LIN {X 0,Y 306.218,Z 83.638,A -85,B 0,C 180,E1 15314.136,E2 15314.136} C_VEL
LIN {X 0,Y 306.221,Z 83.636,A -85,B 0,C 180,E1 15309.585,E2 15309.585} C_VEL
LIN {X 0,Y 306.232,Z 83.637,A -85,B 0,C 180,E1 15305.245,E2 15305.245} C_VEL
LIN {X 0,Y 306.224,Z 83.64,A -85,B 0,C 180,E1 15300.748,E2 15300.748} C_VEL
LIN {X 0,Y 306.21,Z 83.649,A -85,B 0,C 180,E1 15296.255,E2 15296.255} C_VEL
LIN {X 0,Y 306.226,Z 83.648,A -85,B 0,C 180,E1 15291.74,E2 15291.74} C_VEL
LIN {X 0,Y 306.224,Z 83.645,A -85,B 0,C 180,E1 15287.171,E2 15287.171} C_VEL
LIN {X 0,Y 306.206,Z 83.645,A -85,B 0,C 180,E1 15282.713,E2 15282.713} C_VEL
LIN {X 0,Y 306.211,Z 83.626,A -85,B 0,C 180,E1 15278.146,E2 15278.146} C_VEL
LIN {X 0,Y 306.227,Z 83.646,A -85,B 0,C 180,E1 15273.637,E2 15273.637} C_VEL
LIN {X 0,Y 306.201,Z 83.621,A -85,B 0,C 180,E1 15269.158,E2 15269.158} C_VEL
LIN {X 0,Y 306.198,Z 83.63,A -85,B 0,C 180,E1 15264.691,E2 15264.691} C_VEL
LIN {X 0,Y 306.254,Z 83.929,A -85,B 0,C 180,E1 15261.619,E2 15261.619} C_VEL
LIN {X 0,Y 307.429,Z 87.023,A -85,B 0,C 180,E1 15260.879,E2 15260.879} C_VEL
LIN {X 0,Y 312.046,Z 96.934,A -85,B 0,C 180,E1 15258.694,E2 15258.694} C_VEL
LIN {X 0,Y 317.804,Z 111.108,A -85,B 0,C 180,E1 15255.831,E2 15255.831} C_VEL
LIN {X 0,Y 322.826,Z 126.337,A -85,B 0,C 180,E1 15253.034,E2 15253.034} C_VEL
LIN {X 0,Y 325.376,Z 136.231,A -85,B 0,C 180,E1 15251.349,E2 15251.349} C_VEL
LIN {X 0,Y 323.736,Z 169.935,A -85,B 0,C 180,E1 15247.17,E2 15247.17} C_VEL
LIN {X 0,Y 322.19,Z 205.367,A -85,B 0,C 180,E1 15242.891,E2 15242.891} C_VEL
LIN {X 0,Y 322.186,Z 209.699,A -85,B 0,C 180,E1 15242.451,E2 15242.451} C_VEL
LIN {X 0,Y 322.798,Z 215.074,A -85,B 0,C 180,E1 15242.253,E2 15242.253} C_VEL
LIN {X 0,Y 320.257,Z 311.161,A -85,B 0,C 180,E1 15240.104,E2 15240.104} C_VEL
LIN {X 0,Y 320.153,Z 327.939,A -85,B 0,C 180,E1 15239.578,E2 15239.578} C_VEL
LIN {X 0,Y 319.58,Z 341.902,A -85,B 0,C 180,E1 15238.832,E2 15238.832} C_VEL
LIN {X 0,Y 318.545,Z 355.587,A -85,B 0,C 180,E1 15237.78,E2 15237.78} C_VEL
LIN {X 0,Y 317.068,Z 368.764,A -85,B 0,C 180,E1 15236.398,E2 15236.398} C_VEL
LIN {X 0,Y 315.473,Z 380.218,A -85,B 0,C 180,E1 15234.829,E2 15234.829} C_VEL
LIN {X 0,Y 313.629,Z 391.275,A -85,B 0,C 180,E1 15232.887,E2 15232.887} C_VEL
LIN {X 0,Y 311.744,Z 401.04,A -85,B 0,C 180,E1 15230.657,E2 15230.657} C_VEL
LIN {X 0,Y 310.021,Z 409.095,A -85,B 0,C 180,E1 15228.229,E2 15228.229} C_VEL
LIN {X 0,Y 308.649,Z 415.111,A -85,B 0,C 180,E1 15225.788,E2 15225.788} C_VEL
LIN {X 0,Y 307.543,Z 419.693,A -85,B 0,C 180,E1 15223.153,E2 15223.153} C_VEL
LIN {X 0,Y 306.711,Z 422.772,A -85,B 0,C 180,E1 15220.137,E2 15220.137} C_VEL
LIN {X 0,Y 306.28,Z 423.761,A -85,B 0,C 180,E1 15217.124,E2 15217.124} C_VEL
LIN {X 0,Y 306.204,Z 422.716,A -85,B 0,C 180,E1 15214.118,E2 15214.118} C_VEL
LIN {X 0,Y 306.447,Z 419.874,A -85,B 0,C 180,E1 15211.307,E2 15211.307} C_VEL
LIN {X 0,Y 306.968,Z 415.503,A -85,B 0,C 180,E1 15208.692,E2 15208.692} C_VEL
LIN {X 0,Y 307.795,Z 409.247,A -85,B 0,C 180,E1 15206.087,E2 15206.087} C_VEL
LIN {X 0,Y 308.953,Z 400.726,A -85,B 0,C 180,E1 15203.495,E2 15203.495} C_VEL
LIN {X 0,Y 310.21,Z 391.122,A -85,B 0,C 180,E1 15201.286,E2 15201.286} C_VEL
LIN {X 0,Y 311.494,Z 380.394,A -85,B 0,C 180,E1 15199.363,E2 15199.363} C_VEL
LIN {X 0,Y 312.685,Z 368.716,A -85,B 0,C 180,E1 15197.721,E2 15197.721} C_VEL
LIN {X 0,Y 313.807,Z 355.087,A -85,B 0,C 180,E1 15196.267,E2 15196.267} C_VEL
LIN {X 0,Y 314.647,Z 340.308,A -85,B 0,C 180,E1 15195.13,E2 15195.13} C_VEL
LIN {X 0,Y 315.034,Z 325.009,A -85,B 0,C 180,E1 15194.342,E2 15194.342} C_VEL
LIN {X 0,Y 315.24,Z 322.674,A -85,B 0,C 180,E1 15194.17,E2 15194.17} C_VEL
LIN {X 0,Y 316.013,Z 321.401,A -85,B 0,C 180,E1 15193.879,E2 15193.879} C_VEL
LIN {X 0,Y 316.94,Z 321.781,A -85,B 0,C 180,E1 15193.693,E2 15193.693} C_VEL
LIN {X 0,Y 319.234,Z 322.708,A -85,B 0,C 180,E1 15193.439,E2 15193.439} C_VEL
LIN {X 0,Y 317.966,Z 338.659,A -85,B 0,C 180,E1 15192.327,E2 15192.327} C_VEL
LIN {X 0,Y 316.409,Z 352.982,A -85,B 0,C 180,E1 15191.004,E2 15191.004} C_VEL
LIN {X 0,Y 314.606,Z 366.938,A -85,B 0,C 180,E1 15189.342,E2 15189.342} C_VEL
LIN {X 0,Y 312.817,Z 379.43,A -85,B 0,C 180,E1 15187.445,E2 15187.445} C_VEL
LIN {X 0,Y 311.381,Z 388.653,A -85,B 0,C 180,E1 15185.723,E2 15185.723} C_VEL
LIN {X 0,Y 309.626,Z 393.761,A -85,B 0,C 180,E1 15184.686,E2 15184.686} C_VEL
LIN {X 0,Y 303.524,Z 403.055,A -85,B 0,C 180,E1 15182.617,E2 15182.617} C_VEL
LIN {X 0,Y 300.836,Z 407.741,A -85,B 0,C 180,E1 15181.279,E2 15181.279} C_VEL
LIN {X 0,Y 300.384,Z 409.36,A -85,B 0,C 180,E1 15180.736,E2 15180.736} C_VEL
LIN {X 0,Y 299.326,Z 416.103,A -85,B 0,C 180,E1 15177.918,E2 15177.918} C_VEL
LIN {X 0,Y 298.675,Z 420.99,A -85,B 0,C 180,E1 15175.078,E2 15175.078} C_VEL
LIN {X 0,Y 298.375,Z 424.115,A -85,B 0,C 180,E1 15172.175,E2 15172.175} C_VEL
LIN {X 0,Y 298.432,Z 425.598,A -85,B 0,C 180,E1 15169.206,E2 15169.206} C_VEL
LIN {X 0,Y 298.87,Z 425.294,A -85,B 0,C 180,E1 15166.17,E2 15166.17} C_VEL
LIN {X 0,Y 299.771,Z 423.124,A -85,B 0,C 180,E1 15163.074,E2 15163.074} C_VEL
LIN {X 0,Y 301.067,Z 419.248,A -85,B 0,C 180,E1 15160.195,E2 15160.195} C_VEL
LIN {X 0,Y 302.907,Z 413.394,A -85,B 0,C 180,E1 15157.295,E2 15157.295} C_VEL
LIN {X 0,Y 305.079,Z 405.985,A -85,B 0,C 180,E1 15154.651,E2 15154.651} C_VEL
LIN {X 0,Y 307.546,Z 397.131,A -85,B 0,C 180,E1 15152.221,E2 15152.221} C_VEL
LIN {X 0,Y 310.231,Z 386.618,A -85,B 0,C 180,E1 15149.971,E2 15149.971} C_VEL
LIN {X 0,Y 313.092,Z 374.223,A -85,B 0,C 180,E1 15147.885,E2 15147.885} C_VEL
LIN {X 0,Y 315.783,Z 360.648,A -85,B 0,C 180,E1 15146.112,E2 15146.112} C_VEL
LIN {X 0,Y 318.084,Z 346.959,A -85,B 0,C 180,E1 15144.709,E2 15144.709} C_VEL
LIN {X 0,Y 320.126,Z 331.5,A -85,B 0,C 180,E1 15143.512,E2 15143.512} C_VEL
LIN {X 0,Y 321.698,Z 315.374,A -85,B 0,C 180,E1 15142.606,E2 15142.606} C_VEL
LIN {X 0,Y 322.948,Z 294.587,A -85,B 0,C 180,E1 15141.877,E2 15141.877} C_VEL
LIN {X 0,Y 327.686,Z 217.917,A -85,B 0,C 180,E1 15139.693,E2 15139.693} C_VEL
LIN {X 0,Y 323.711,Z 190.896,A -85,B 0,C 180,E1 15138.038,E2 15138.038} C_VEL
LIN {X 0,Y 320.283,Z 171.007,A -85,B 0,C 180,E1 15136.585,E2 15136.585} C_VEL
LIN {X 0,Y 323.837,Z 155.783,A -85,B 0,C 180,E1 15133.663,E2 15133.663} C_VEL
LIN {X 0,Y 321.635,Z 144.592,A -85,B 0,C 180,E1 15130.388,E2 15130.388} C_VEL
LIN {X 0,Y 319.074,Z 134.629,A -85,B 0,C 180,E1 15127.02,E2 15127.02} C_VEL
LIN {X 0,Y 316.628,Z 126.45,A -85,B 0,C 180,E1 15123.803,E2 15123.803} C_VEL
LIN {X 0,Y 314.2,Z 119.063,A -85,B 0,C 180,E1 15120.365,E2 15120.365} C_VEL
LIN {X 0,Y 312.239,Z 114.196,A -85,B 0,C 180,E1 15117.567,E2 15117.567} C_VEL
LIN {X 0,Y 311.17,Z 111.425,A -85,B 0,C 180,E1 15115.762,E2 15115.762} C_VEL
LIN {X 0,Y 309.858,Z 108.044,A -85,B 0,C 180,E1 15113.143,E2 15113.143} C_VEL
LIN {X 0,Y 308.302,Z 104.197,A -85,B 0,C 180,E1 15108.969,E2 15108.969} C_VEL
LIN {X 0,Y 307.15,Z 102.355,A -85,B 0,C 180,E1 15103.937,E2 15103.937} C_VEL
LIN {X 0,Y 307.285,Z 102.523,A -85,B 0,C 180,E1 15100.023,E2 15100.023} C_VEL
LIN {X 0,Y 308.962,Z 104.848,A -85,B 0,C 180,E1 15094.917,E2 15094.917} C_VEL
LIN {X 0,Y 311.201,Z 109.842,A -85,B 0,C 180,E1 15090.345,E2 15090.345} C_VEL
LIN {X 0,Y 313.233,Z 114.532,A -85,B 0,C 180,E1 15087.354,E2 15087.354} C_VEL
LIN {X 0,Y 315.016,Z 118.627,A -85,B 0,C 180,E1 15085.158,E2 15085.158} C_VEL
LIN {X 0,Y 317.64,Z 124.79,A -85,B 0,C 180,E1 15082.362,E2 15082.362} C_VEL
LIN {X 0,Y 321.226,Z 134.301,A -85,B 0,C 180,E1 15078.874,E2 15078.874} C_VEL
LIN {X 0,Y 324.75,Z 144.909,A -85,B 0,C 180,E1 15075.662,E2 15075.662} C_VEL
LIN {X 0,Y 328.156,Z 157.046,A -85,B 0,C 180,E1 15072.565,E2 15072.565} C_VEL
LIN {X 0,Y 328.381,Z 158.338,A -85,B 0,C 180,E1 15072.278,E2 15072.278} C_VEL
LIN {X 0,Y 326.983,Z 164.325,A -85,B 0,C 180,E1 15071.492,E2 15071.492} C_VEL
LIN {X 0,Y 329.661,Z 192.112,A -85,B 0,C 180,E1 15070.189,E2 15070.189} C_VEL
LIN {X 0,Y 329.69,Z 198.596,A -85,B 0,C 180,E1 15069.987,E2 15069.987} C_VEL
LIN {X 0,Y 324.108,Z 330.652,A -85,B 0,C 180,E1 15067,E2 15067} C_VEL
LIN {X 0,Y 322.996,Z 351.571,A -85,B 0,C 180,E1 15066.447,E2 15066.447} C_VEL
LIN {X 0,Y 321.026,Z 369.794,A -85,B 0,C 180,E1 15065.677,E2 15065.677} C_VEL
LIN {X 0,Y 318.428,Z 386.883,A -85,B 0,C 180,E1 15064.635,E2 15064.635} C_VEL
LIN {X 0,Y 315.355,Z 403.595,A -85,B 0,C 180,E1 15063.266,E2 15063.266} C_VEL
LIN {X 0,Y 311.891,Z 420.167,A -85,B 0,C 180,E1 15061.504,E2 15061.504} C_VEL
LIN {X 0,Y 308.53,Z 435.036,A -85,B 0,C 180,E1 15059.512,E2 15059.512} C_VEL
LIN {X 0,Y 305.249,Z 448.999,A -85,B 0,C 180,E1 15057.191,E2 15057.191} C_VEL
LIN {X 0,Y 302.216,Z 462.009,A -85,B 0,C 180,E1 15054.521,E2 15054.521} C_VEL
LIN {X 0,Y 299.688,Z 473.731,A -85,B 0,C 180,E1 15051.532,E2 15051.532} C_VEL
LIN {X 0,Y 297.903,Z 483.696,A -85,B 0,C 180,E1 15048.392,E2 15048.392} C_VEL
LIN {X 0,Y 296.829,Z 492.632,A -85,B 0,C 180,E1 15044.834,E2 15044.834} C_VEL
LIN {X 0,Y 296.583,Z 499.123,A -85,B 0,C 180,E1 15041.474,E2 15041.474} C_VEL
LIN {X 0,Y 296.941,Z 504.12,A -85,B 0,C 180,E1 15037.937,E2 15037.937} C_VEL
LIN {X 0,Y 297.552,Z 507.104,A -85,B 0,C 180,E1 15034.627,E2 15034.627} C_VEL
LIN {X 0,Y 298.008,Z 508.377,A -85,B 0,C 180,E1 15031.539,E2 15031.539} C_VEL
LIN {X 0,Y 298.055,Z 508.203,A -85,B 0,C 180,E1 15028.656,E2 15028.656} C_VEL
LIN {X 0,Y 297.673,Z 506.535,A -85,B 0,C 180,E1 15025.571,E2 15025.571} C_VEL
LIN {X 0,Y 297.132,Z 503.314,A -85,B 0,C 180,E1 15022.461,E2 15022.461} C_VEL
LIN {X 0,Y 296.743,Z 498.122,A -85,B 0,C 180,E1 15019.125,E2 15019.125} C_VEL
LIN {X 0,Y 296.849,Z 491.021,A -85,B 0,C 180,E1 15015.768,E2 15015.768} C_VEL
LIN {X 0,Y 297.621,Z 481.81,A -85,B 0,C 180,E1 15012.403,E2 15012.403} C_VEL
LIN {X 0,Y 298.972,Z 471.647,A -85,B 0,C 180,E1 15009.444,E2 15009.444} C_VEL
LIN {X 0,Y 300.853,Z 460.093,A -85,B 0,C 180,E1 15006.706,E2 15006.706} C_VEL
LIN {X 0,Y 303.17,Z 447.087,A -85,B 0,C 180,E1 15004.195,E2 15004.195} C_VEL
LIN {X 0,Y 305.808,Z 432.438,A -85,B 0,C 180,E1 15001.915,E2 15001.915} C_VEL
LIN {X 0,Y 308.392,Z 417.575,A -85,B 0,C 180,E1 15000.049,E2 15000.049} C_VEL
LIN {X 0,Y 311.025,Z 401.011,A -85,B 0,C 180,E1 14998.401,E2 14998.401} C_VEL
LIN {X 0,Y 313.395,Z 383.904,A -85,B 0,C 180,E1 14997.097,E2 14997.097} C_VEL
LIN {X 0,Y 315.377,Z 366.084,A -85,B 0,C 180,E1 14996.106,E2 14996.106} C_VEL
LIN {X 0,Y 316.7,Z 347.608,A -85,B 0,C 180,E1 14995.417,E2 14995.417} C_VEL
LIN {X 0,Y 322.005,Z 178.475,A -85,B 0,C 180,E1 14991.663,E2 14991.663} C_VEL
LIN {X 0,Y 321.492,Z 158.885,A -85,B 0,C 180,E1 14991.083,E2 14991.083} C_VEL
LIN {X 0,Y 323.297,Z 143.638,A -85,B 0,C 180,E1 14989.9,E2 14989.9} C_VEL
LIN {X 0,Y 314.968,Z 122.157,A -85,B 0,C 180,E1 14986.897,E2 14986.897} C_VEL
LIN {X 0,Y 306.931,Z 103.52,A -85,B 0,C 180,E1 14983.937,E2 14983.937} C_VEL
LIN {X 0,Y 299.48,Z 87.935,A -85,B 0,C 180,E1 14981.125,E2 14981.125} C_VEL
LIN {X 0,Y 298.366,Z 85.034,A -85,B 0,C 180,E1 14980.55,E2 14980.55} C_VEL
LIN {X 0,Y 298.295,Z 84.644,A -85,B 0,C 180,E1 14979.808,E2 14979.808} C_VEL
LIN {X 0,Y 298.29,Z 84.632,A -85,B 0,C 180,E1 14975.131,E2 14975.131} C_VEL
LIN {X 0,Y 298.304,Z 84.636,A -85,B 0,C 180,E1 14970.529,E2 14970.529} C_VEL
LIN {X 0,Y 298.288,Z 84.642,A -85,B 0,C 180,E1 14966.047,E2 14966.047} C_VEL
LIN {X 0,Y 298.289,Z 84.641,A -85,B 0,C 180,E1 14961.43,E2 14961.43} C_VEL
LIN {X 0,Y 298.297,Z 84.64,A -85,B 0,C 180,E1 14956.954,E2 14956.954} C_VEL
LIN {X 0,Y 298.29,Z 84.638,A -85,B 0,C 180,E1 14952.584,E2 14952.584} C_VEL
LIN {X 0,Y 298.279,Z 84.638,A -85,B 0,C 180,E1 14947.899,E2 14947.899} C_VEL
LIN {X 0,Y 298.29,Z 84.633,A -85,B 0,C 180,E1 14943.266,E2 14943.266} C_VEL
LIN {X 0,Y 298.286,Z 84.628,A -85,B 0,C 180,E1 14938.847,E2 14938.847} C_VEL
LIN {X 0,Y 298.27,Z 84.632,A -85,B 0,C 180,E1 14934.228,E2 14934.228} C_VEL
LIN {X 0,Y 298.282,Z 84.628,A -85,B 0,C 180,E1 14929.766,E2 14929.766} C_VEL
LIN {X 0,Y 298.29,Z 84.629,A -85,B 0,C 180,E1 14925.241,E2 14925.241} C_VEL
LIN {X 0,Y 298.267,Z 84.64,A -85,B 0,C 180,E1 14920.617,E2 14920.617} C_VEL
LIN {X 0,Y 298.275,Z 84.594,A -85,B 0,C 180,E1 14916.07,E2 14916.07} C_VEL
LIN {X 0,Y 298.285,Z 84.622,A -85,B 0,C 180,E1 14911.576,E2 14911.576} C_VEL
LIN {X 0,Y 298.263,Z 84.646,A -85,B 0,C 180,E1 14907.107,E2 14907.107} C_VEL
LIN {X 0,Y 298.285,Z 84.823,A -85,B 0,C 180,E1 14903.05,E2 14903.05} C_VEL
LIN {X 0,Y 299.159,Z 87.431,A -85,B 0,C 180,E1 14902.379,E2 14902.379} C_VEL
LIN {X 0,Y 300.565,Z 90.006,A -85,B 0,C 180,E1 14901.724,E2 14901.724} C_VEL
LIN {X 0,Y 306.143,Z 102.165,A -85,B 0,C 180,E1 14898.969,E2 14898.969} C_VEL
LIN {X 0,Y 311.601,Z 115.952,A -85,B 0,C 180,E1 14896.124,E2 14896.124} C_VEL
LIN {X 0,Y 316.602,Z 131.405,A -85,B 0,C 180,E1 14893.257,E2 14893.257} C_VEL
LIN {X 0,Y 318.588,Z 138.968,A -85,B 0,C 180,E1 14891.943,E2 14891.943} C_VEL
LIN {X 0,Y 316.728,Z 174.086,A -85,B 0,C 180,E1 14887.534,E2 14887.534} C_VEL
LIN {X 0,Y 315.112,Z 210.08,A -85,B 0,C 180,E1 14883.186,E2 14883.186} C_VEL
LIN {X 0,Y 315.824,Z 216.202,A -85,B 0,C 180,E1 14882.945,E2 14882.945} C_VEL
LIN {X 0,Y 313.162,Z 311.56,A -85,B 0,C 180,E1 14880.769,E2 14880.769} C_VEL
LIN {X 0,Y 313.042,Z 328.708,A -85,B 0,C 180,E1 14880.227,E2 14880.227} C_VEL
LIN {X 0,Y 312.47,Z 342.308,A -85,B 0,C 180,E1 14879.498,E2 14879.498} C_VEL
LIN {X 0,Y 311.3,Z 356.975,A -85,B 0,C 180,E1 14878.35,E2 14878.35} C_VEL
LIN {X 0,Y 309.679,Z 370.641,A -85,B 0,C 180,E1 14876.871,E2 14876.871} C_VEL
LIN {X 0,Y 307.907,Z 382.491,A -85,B 0,C 180,E1 14875.174,E2 14875.174} C_VEL
LIN {X 0,Y 306.065,Z 392.819,A -85,B 0,C 180,E1 14873.282,E2 14873.282} C_VEL
LIN {X 0,Y 304.091,Z 402.488,A -85,B 0,C 180,E1 14871,E2 14871} C_VEL
LIN {X 0,Y 302.286,Z 410.469,A -85,B 0,C 180,E1 14868.512,E2 14868.512} C_VEL
LIN {X 0,Y 300.748,Z 416.791,A -85,B 0,C 180,E1 14865.818,E2 14865.818} C_VEL
LIN {X 0,Y 299.61,Z 421.153,A -85,B 0,C 180,E1 14863.115,E2 14863.115} C_VEL
LIN {X 0,Y 298.805,Z 423.925,A -85,B 0,C 180,E1 14860.214,E2 14860.214} C_VEL
LIN {X 0,Y 298.354,Z 424.856,A -85,B 0,C 180,E1 14857.121,E2 14857.121} C_VEL
LIN {X 0,Y 298.28,Z 423.753,A -85,B 0,C 180,E1 14854.035,E2 14854.035} C_VEL
LIN {X 0,Y 298.542,Z 420.842,A -85,B 0,C 180,E1 14851.15,E2 14851.15} C_VEL
LIN {X 0,Y 299.097,Z 416.397,A -85,B 0,C 180,E1 14848.466,E2 14848.466} C_VEL
LIN {X 0,Y 299.977,Z 410.066,A -85,B 0,C 180,E1 14845.793,E2 14845.793} C_VEL
LIN {X 0,Y 301.102,Z 402.148,A -85,B 0,C 180,E1 14843.324,E2 14843.324} C_VEL
LIN {X 0,Y 302.41,Z 392.647,A -85,B 0,C 180,E1 14841.059,E2 14841.059} C_VEL
LIN {X 0,Y 303.748,Z 382.05,A -85,B 0,C 180,E1 14839.088,E2 14839.088} C_VEL
LIN {X 0,Y 305.064,Z 369.787,A -85,B 0,C 180,E1 14837.314,E2 14837.314} C_VEL
LIN {X 0,Y 306.24,Z 356.15,A -85,B 0,C 180,E1 14835.825,E2 14835.825} C_VEL
LIN {X 0,Y 307.124,Z 341.358,A -85,B 0,C 180,E1 14834.661,E2 14834.661} C_VEL
LIN {X 0,Y 307.553,Z 332.982,A -85,B 0,C 180,E1 14834.107,E2 14834.107} C_VEL
LIN {X 0,Y 308.443,Z 331.887,A -85,B 0,C 180,E1 14833.763,E2 14833.763} C_VEL
LIN {X 0,Y 311.174,Z 333.159,A -85,B 0,C 180,E1 14833.355,E2 14833.355} C_VEL
LIN {X 0,Y 309.531,Z 348.896,A -85,B 0,C 180,E1 14832.009,E2 14832.009} C_VEL
LIN {X 0,Y 307.639,Z 363.677,A -85,B 0,C 180,E1 14830.352,E2 14830.352} C_VEL
LIN {X 0,Y 305.596,Z 377.731,A -85,B 0,C 180,E1 14828.301,E2 14828.301} C_VEL
LIN {X 0,Y 303.681,Z 389.594,A -85,B 0,C 180,E1 14826.088,E2 14826.088} C_VEL
LIN {X 0,Y 301.964,Z 399.884,A -85,B 0,C 180,E1 14823.659,E2 14823.659} C_VEL
LIN {X 0,Y 300.472,Z 408.792,A -85,B 0,C 180,E1 14820.932,E2 14820.932} C_VEL
LIN {X 0,Y 300.384,Z 409.36,A -85,B 0,C 180,E1 14820.736,E2 14820.736} C_VEL
LIN {X 0,Y 298.873,Z 412.989,A -85,B 0,C 180,E1 14819.453,E2 14819.453} C_VEL
LIN {X 0,Y 294.088,Z 418.356,A -85,B 0,C 180,E1 14817.258,E2 14817.258} C_VEL
LIN {X 0,Y 291.155,Z 421.554,A -85,B 0,C 180,E1 14815.481,E2 14815.481} C_VEL
LIN {X 0,Y 290.67,Z 422.702,A -85,B 0,C 180,E1 14814.639,E2 14814.639} C_VEL
LIN {X 0,Y 290.43,Z 425.743,A -85,B 0,C 180,E1 14811.454,E2 14811.454} C_VEL
LIN {X 0,Y 290.597,Z 426.821,A -85,B 0,C 180,E1 14808.3,E2 14808.3} C_VEL
LIN {X 0,Y 291.176,Z 426.156,A -85,B 0,C 180,E1 14805.255,E2 14805.255} C_VEL
LIN {X 0,Y 292.151,Z 423.829,A -85,B 0,C 180,E1 14802.332,E2 14802.332} C_VEL
LIN {X 0,Y 293.674,Z 419.566,A -85,B 0,C 180,E1 14799.292,E2 14799.292} C_VEL
LIN {X 0,Y 295.672,Z 413.576,A -85,B 0,C 180,E1 14796.405,E2 14796.405} C_VEL
LIN {X 0,Y 298.186,Z 405.572,A -85,B 0,C 180,E1 14793.592,E2 14793.592} C_VEL
LIN {X 0,Y 300.902,Z 396.224,A -85,B 0,C 180,E1 14791.101,E2 14791.101} C_VEL
LIN {X 0,Y 303.732,Z 385.585,A -85,B 0,C 180,E1 14788.877,E2 14788.877} C_VEL
LIN {X 0,Y 306.49,Z 374.05,A -85,B 0,C 180,E1 14786.966,E2 14786.966} C_VEL
LIN {X 0,Y 309.467,Z 359.746,A -85,B 0,C 180,E1 14785.102,E2 14785.102} C_VEL
LIN {X 0,Y 311.913,Z 345.474,A -85,B 0,C 180,E1 14783.672,E2 14783.672} C_VEL
LIN {X 0,Y 314.095,Z 329.395,A -85,B 0,C 180,E1 14782.458,E2 14782.458} C_VEL
LIN {X 0,Y 315.67,Z 312.422,A -85,B 0,C 180,E1 14781.569,E2 14781.569} C_VEL
LIN {X 0,Y 317.627,Z 281.324,A -85,B 0,C 180,E1 14780.578,E2 14780.578} C_VEL
LIN {X 0,Y 321.613,Z 219.163,A -85,B 0,C 180,E1 14778.782,E2 14778.782} C_VEL
LIN {X 0,Y 317.859,Z 192.52,A -85,B 0,C 180,E1 14777.081,E2 14777.081} C_VEL
LIN {X 0,Y 314.18,Z 170.966,A -85,B 0,C 180,E1 14775.455,E2 14775.455} C_VEL
LIN {X 0,Y 317.08,Z 159.096,A -85,B 0,C 180,E1 14773.123,E2 14773.123} C_VEL
LIN {X 0,Y 315.055,Z 148.38,A -85,B 0,C 180,E1 14769.868,E2 14769.868} C_VEL
LIN {X 0,Y 312.512,Z 138.076,A -85,B 0,C 180,E1 14766.245,E2 14766.245} C_VEL
LIN {X 0,Y 309.93,Z 129.366,A -85,B 0,C 180,E1 14762.589,E2 14762.589} C_VEL
LIN {X 0,Y 307.785,Z 123.166,A -85,B 0,C 180,E1 14759.442,E2 14759.442} C_VEL
LIN {X 0,Y 306.027,Z 117.882,A -85,B 0,C 180,E1 14756.254,E2 14756.254} C_VEL
LIN {X 0,Y 304.313,Z 113.734,A -85,B 0,C 180,E1 14752.87,E2 14752.87} C_VEL
LIN {X 0,Y 302.929,Z 110.091,A -85,B 0,C 180,E1 14748.771,E2 14748.771} C_VEL
LIN {X 0,Y 301.922,Z 108.386,A -85,B 0,C 180,E1 14743.651,E2 14743.651} C_VEL
LIN {X 0,Y 302.176,Z 108.736,A -85,B 0,C 180,E1 14739.67,E2 14739.67} C_VEL
LIN {X 0,Y 303.784,Z 111.056,A -85,B 0,C 180,E1 14734.841,E2 14734.841} C_VEL
LIN {X 0,Y 305.898,Z 115.909,A -85,B 0,C 180,E1 14730.396,E2 14730.396} C_VEL
LIN {X 0,Y 307.724,Z 120.203,A -85,B 0,C 180,E1 14727.58,E2 14727.58} C_VEL
LIN {X 0,Y 309.665,Z 124.824,A -85,B 0,C 180,E1 14725.098,E2 14725.098} C_VEL
LIN {X 0,Y 312.169,Z 131.034,A -85,B 0,C 180,E1 14722.283,E2 14722.283} C_VEL
LIN {X 0,Y 315.429,Z 139.952,A -85,B 0,C 180,E1 14718.976,E2 14718.976} C_VEL
LIN {X 0,Y 318.791,Z 150.454,A -85,B 0,C 180,E1 14715.746,E2 14715.746} C_VEL
LIN {X 0,Y 321.704,Z 161.505,A -85,B 0,C 180,E1 14712.896,E2 14712.896} C_VEL
LIN {X 0,Y 321.066,Z 164.544,A -85,B 0,C 180,E1 14712.516,E2 14712.516} C_VEL
LIN {X 0,Y 323.554,Z 191.512,A -85,B 0,C 180,E1 14711.182,E2 14711.182} C_VEL
LIN {X 0,Y 323.746,Z 198.251,A -85,B 0,C 180,E1 14710.934,E2 14710.934} C_VEL
LIN {X 0,Y 316.998,Z 346.321,A -85,B 0,C 180,E1 14707.479,E2 14707.479} C_VEL
LIN {X 0,Y 315.136,Z 364.811,A -85,B 0,C 180,E1 14706.754,E2 14706.754} C_VEL
LIN {X 0,Y 312.668,Z 381.422,A -85,B 0,C 180,E1 14705.818,E2 14705.818} C_VEL
LIN {X 0,Y 309.617,Z 398.158,A -85,B 0,C 180,E1 14704.536,E2 14704.536} C_VEL
LIN {X 0,Y 306.226,Z 414.206,A -85,B 0,C 180,E1 14702.933,E2 14702.933} C_VEL
LIN {X 0,Y 302.687,Z 429.303,A -85,B 0,C 180,E1 14701.019,E2 14701.019} C_VEL
LIN {X 0,Y 299.026,Z 443.988,A -85,B 0,C 180,E1 14698.675,E2 14698.675} C_VEL
LIN {X 0,Y 295.724,Z 457.159,A -85,B 0,C 180,E1 14696.076,E2 14696.076} C_VEL
LIN {X 0,Y 292.831,Z 469.263,A -85,B 0,C 180,E1 14693.121,E2 14693.121} C_VEL
LIN {X 0,Y 290.623,Z 479.85,A -85,B 0,C 180,E1 14689.915,E2 14689.915} C_VEL
LIN {X 0,Y 289.191,Z 488.934,A -85,B 0,C 180,E1 14686.471,E2 14686.471} C_VEL
LIN {X 0,Y 288.614,Z 496.386,A -85,B 0,C 180,E1 14682.811,E2 14682.811} C_VEL
LIN {X 0,Y 288.785,Z 501.85,A -85,B 0,C 180,E1 14679.166,E2 14679.166} C_VEL
LIN {X 0,Y 289.391,Z 505.332,A -85,B 0,C 180,E1 14675.704,E2 14675.704} C_VEL
LIN {X 0,Y 289.953,Z 507.042,A -85,B 0,C 180,E1 14672.571,E2 14672.571} C_VEL
LIN {X 0,Y 290.173,Z 507.299,A -85,B 0,C 180,E1 14669.607,E2 14669.607} C_VEL
LIN {X 0,Y 289.911,Z 506.154,A -85,B 0,C 180,E1 14666.64,E2 14666.64} C_VEL
LIN {X 0,Y 289.357,Z 503.445,A -85,B 0,C 180,E1 14663.454,E2 14663.454} C_VEL
LIN {X 0,Y 288.847,Z 498.832,A -85,B 0,C 180,E1 14660.035,E2 14660.035} C_VEL
LIN {X 0,Y 288.794,Z 492.358,A -85,B 0,C 180,E1 14656.589,E2 14656.589} C_VEL
LIN {X 0,Y 289.371,Z 483.918,A -85,B 0,C 180,E1 14653.159,E2 14653.159} C_VEL
LIN {X 0,Y 290.585,Z 474.343,A -85,B 0,C 180,E1 14650.086,E2 14650.086} C_VEL
LIN {X 0,Y 292.48,Z 462.627,A -85,B 0,C 180,E1 14647.065,E2 14647.065} C_VEL
LIN {X 0,Y 294.735,Z 450.263,A -85,B 0,C 180,E1 14644.472,E2 14644.472} C_VEL
LIN {X 0,Y 297.436,Z 435.961,A -85,B 0,C 180,E1 14642.037,E2 14642.037} C_VEL
LIN {X 0,Y 300.257,Z 420.604,A -85,B 0,C 180,E1 14639.936,E2 14639.936} C_VEL
LIN {X 0,Y 302.929,Z 404.953,A -85,B 0,C 180,E1 14638.236,E2 14638.236} C_VEL
LIN {X 0,Y 305.378,Z 388.657,A -85,B 0,C 180,E1 14636.856,E2 14636.856} C_VEL
LIN {X 0,Y 307.602,Z 370.716,A -85,B 0,C 180,E1 14635.735,E2 14635.735} C_VEL
LIN {X 0,Y 309.172,Z 352.612,A -85,B 0,C 180,E1 14634.956,E2 14634.956} C_VEL
LIN {X 0,Y 310.134,Z 327.851,A -85,B 0,C 180,E1 14634.322,E2 14634.322} C_VEL
LIN {X 0,Y 315.038,Z 179.291,A -85,B 0,C 180,E1 14630.971,E2 14630.971} C_VEL
LIN {X 0,Y 314.622,Z 158.089,A -85,B 0,C 180,E1 14630.302,E2 14630.302} C_VEL
LIN {X 0,Y 316.097,Z 146.113,A -85,B 0,C 180,E1 14629.34,E2 14629.34} C_VEL
LIN {X 0,Y 307.764,Z 124.504,A -85,B 0,C 180,E1 14626.215,E2 14626.215} C_VEL
LIN {X 0,Y 299.01,Z 104.371,A -85,B 0,C 180,E1 14622.881,E2 14622.881} C_VEL
LIN {X 0,Y 291.934,Z 89.484,A -85,B 0,C 180,E1 14620.082,E2 14620.082} C_VEL
LIN {X 0,Y 290.433,Z 86.152,A -85,B 0,C 180,E1 14619.388,E2 14619.388} C_VEL
LIN {X 0,Y 290.362,Z 85.623,A -85,B 0,C 180,E1 14618.905,E2 14618.905} C_VEL
LIN {X 0,Y 290.357,Z 85.625,A -85,B 0,C 180,E1 14614.145,E2 14614.145} C_VEL
LIN {X 0,Y 290.351,Z 85.63,A -85,B 0,C 180,E1 14609.402,E2 14609.402} C_VEL
LIN {X 0,Y 290.358,Z 85.623,A -85,B 0,C 180,E1 14604.841,E2 14604.841} C_VEL
LIN {X 0,Y 290.351,Z 85.624,A -85,B 0,C 180,E1 14600.353,E2 14600.353} C_VEL
LIN {X 0,Y 290.344,Z 85.624,A -85,B 0,C 180,E1 14595.581,E2 14595.581} C_VEL
LIN {X 0,Y 290.354,Z 85.623,A -85,B 0,C 180,E1 14590.917,E2 14590.917} C_VEL
LIN {X 0,Y 290.339,Z 85.627,A -85,B 0,C 180,E1 14586.326,E2 14586.326} C_VEL
LIN {X 0,Y 290.348,Z 85.628,A -85,B 0,C 180,E1 14581.578,E2 14581.578} C_VEL
LIN {X 0,Y 290.347,Z 85.63,A -85,B 0,C 180,E1 14576.989,E2 14576.989} C_VEL
LIN {X 0,Y 290.332,Z 85.632,A -85,B 0,C 180,E1 14572.281,E2 14572.281} C_VEL
LIN {X 0,Y 290.348,Z 85.628,A -85,B 0,C 180,E1 14567.672,E2 14567.672} C_VEL
LIN {X 0,Y 290.343,Z 85.625,A -85,B 0,C 180,E1 14563.185,E2 14563.185} C_VEL
LIN {X 0,Y 290.324,Z 85.611,A -85,B 0,C 180,E1 14558.588,E2 14558.588} C_VEL
LIN {X 0,Y 290.342,Z 85.611,A -85,B 0,C 180,E1 14553.997,E2 14553.997} C_VEL
LIN {X 0,Y 290.344,Z 85.592,A -85,B 0,C 180,E1 14549.587,E2 14549.587} C_VEL
LIN {X 0,Y 290.32,Z 85.62,A -85,B 0,C 180,E1 14544.89,E2 14544.89} C_VEL
LIN {X 0,Y 290.402,Z 86.088,A -85,B 0,C 180,E1 14544.417,E2 14544.417} C_VEL
LIN {X 0,Y 292.148,Z 89.784,A -85,B 0,C 180,E1 14543.451,E2 14543.451} C_VEL
LIN {X 0,Y 297.834,Z 101.678,A -85,B 0,C 180,E1 14540.542,E2 14540.542} C_VEL
LIN {X 0,Y 303.541,Z 115.56,A -85,B 0,C 180,E1 14537.525,E2 14537.525} C_VEL
LIN {X 0,Y 308.446,Z 129.845,A -85,B 0,C 180,E1 14534.7,E2 14534.7} C_VEL
LIN {X 0,Y 311.807,Z 142.278,A -85,B 0,C 180,E1 14532.478,E2 14532.478} C_VEL
LIN {X 0,Y 309.768,Z 178.097,A -85,B 0,C 180,E1 14527.941,E2 14527.941} C_VEL
LIN {X 0,Y 308.184,Z 211.152,A -85,B 0,C 180,E1 14523.917,E2 14523.917} C_VEL
LIN {X 0,Y 308.902,Z 217.32,A -85,B 0,C 180,E1 14523.669,E2 14523.669} C_VEL
LIN {X 0,Y 306.111,Z 311.998,A -85,B 0,C 180,E1 14521.464,E2 14521.464} C_VEL
LIN {X 0,Y 305.974,Z 329.487,A -85,B 0,C 180,E1 14520.905,E2 14520.905} C_VEL
LIN {X 0,Y 305.34,Z 343.61,A -85,B 0,C 180,E1 14520.133,E2 14520.133} C_VEL
LIN {X 0,Y 304.113,Z 358.137,A -85,B 0,C 180,E1 14518.969,E2 14518.969} C_VEL
LIN {X 0,Y 302.415,Z 371.743,A -85,B 0,C 180,E1 14517.464,E2 14517.464} C_VEL
LIN {X 0,Y 300.55,Z 383.594,A -85,B 0,C 180,E1 14515.729,E2 14515.729} C_VEL
LIN {X 0,Y 298.707,Z 393.474,A -85,B 0,C 180,E1 14513.89,E2 14513.89} C_VEL
LIN {X 0,Y 296.612,Z 403.239,A -85,B 0,C 180,E1 14511.555,E2 14511.555} C_VEL
LIN {X 0,Y 294.688,Z 411.294,A -85,B 0,C 180,E1 14509.007,E2 14509.007} C_VEL
LIN {X 0,Y 293.144,Z 417.31,A -85,B 0,C 180,E1 14506.443,E2 14506.443} C_VEL
LIN {X 0,Y 291.895,Z 421.89,A -85,B 0,C 180,E1 14503.67,E2 14503.67} C_VEL
LIN {X 0,Y 290.943,Z 424.967,A -85,B 0,C 180,E1 14500.493,E2 14500.493} C_VEL
LIN {X 0,Y 290.446,Z 425.952,A -85,B 0,C 180,E1 14497.316,E2 14497.316} C_VEL
LIN {X 0,Y 290.347,Z 424.903,A -85,B 0,C 180,E1 14494.146,E2 14494.146} C_VEL
LIN {X 0,Y 290.608,Z 422.057,A -85,B 0,C 180,E1 14491.181,E2 14491.181} C_VEL
LIN {X 0,Y 291.179,Z 417.682,A -85,B 0,C 180,E1 14488.424,E2 14488.424} C_VEL
LIN {X 0,Y 292.087,Z 411.421,A -85,B 0,C 180,E1 14485.68,E2 14485.68} C_VEL
LIN {X 0,Y 293.36,Z 402.892,A -85,B 0,C 180,E1 14482.951,E2 14482.951} C_VEL
LIN {X 0,Y 294.74,Z 393.281,A -85,B 0,C 180,E1 14480.627,E2 14480.627} C_VEL
LIN {X 0,Y 296.148,Z 382.542,A -85,B 0,C 180,E1 14478.607,E2 14478.607} C_VEL
LIN {X 0,Y 297.458,Z 370.85,A -85,B 0,C 180,E1 14476.885,E2 14476.885} C_VEL
LIN {X 0,Y 298.698,Z 357.104,A -85,B 0,C 180,E1 14475.35,E2 14475.35} C_VEL
LIN {X 0,Y 299.815,Z 341.36,A -85,B 0,C 180,E1 14474.029,E2 14474.029} C_VEL
LIN {X 0,Y 300.709,Z 340.513,A -85,B 0,C 180,E1 14473.681,E2 14473.681} C_VEL
LIN {X 0,Y 303.031,Z 341.513,A -85,B 0,C 180,E1 14473.317,E2 14473.317} C_VEL
LIN {X 0,Y 301.235,Z 356.539,A -85,B 0,C 180,E1 14471.819,E2 14471.819} C_VEL
LIN {X 0,Y 299.308,Z 370.123,A -85,B 0,C 180,E1 14470.077,E2 14470.077} C_VEL
LIN {X 0,Y 297.183,Z 383.607,A -85,B 0,C 180,E1 14467.862,E2 14467.862} C_VEL
LIN {X 0,Y 295.237,Z 394.889,A -85,B 0,C 180,E1 14465.488,E2 14465.488} C_VEL
LIN {X 0,Y 293.554,Z 404.522,A -85,B 0,C 180,E1 14462.919,E2 14462.919} C_VEL
LIN {X 0,Y 292.119,Z 412.888,A -85,B 0,C 180,E1 14459.994,E2 14459.994} C_VEL
LIN {X 0,Y 291.172,Z 418.909,A -85,B 0,C 180,E1 14457.141,E2 14457.141} C_VEL
LIN {X 0,Y 290.67,Z 422.702,A -85,B 0,C 180,E1 14454.639,E2 14454.639} C_VEL
LIN {X 0,Y 289.517,Z 424.489,A -85,B 0,C 180,E1 14453.163,E2 14453.163} C_VEL
LIN {X 0,Y 285.191,Z 426.956,A -85,B 0,C 180,E1 14450.553,E2 14450.553} C_VEL
LIN {X 0,Y 282.905,Z 427.906,A -85,B 0,C 180,E1 14448.586,E2 14448.586} C_VEL
LIN {X 0,Y 282.746,Z 427.98,A -85,B 0,C 180,E1 14447.797,E2 14447.797} C_VEL
LIN {X 0,Y 283.381,Z 427.233,A -85,B 0,C 180,E1 14444.83,E2 14444.83} C_VEL
LIN {X 0,Y 284.582,Z 424.517,A -85,B 0,C 180,E1 14441.55,E2 14441.55} C_VEL
LIN {X 0,Y 286.303,Z 420.057,A -85,B 0,C 180,E1 14438.436,E2 14438.436} C_VEL
LIN {X 0,Y 288.625,Z 413.456,A -85,B 0,C 180,E1 14435.347,E2 14435.347} C_VEL
LIN {X 0,Y 291.259,Z 405.517,A -85,B 0,C 180,E1 14432.614,E2 14432.614} C_VEL
LIN {X 0,Y 294.358,Z 395.383,A -85,B 0,C 180,E1 14429.956,E2 14429.956} C_VEL
LIN {X 0,Y 297.277,Z 384.891,A -85,B 0,C 180,E1 14427.8,E2 14427.8} C_VEL
LIN {X 0,Y 300.582,Z 371.532,A -85,B 0,C 180,E1 14425.649,E2 14425.649} C_VEL
LIN {X 0,Y 303.398,Z 358.143,A -85,B 0,C 180,E1 14423.974,E2 14423.974} C_VEL
LIN {X 0,Y 305.997,Z 343.234,A -85,B 0,C 180,E1 14422.528,E2 14422.528} C_VEL
LIN {X 0,Y 308.075,Z 327.652,A -85,B 0,C 180,E1 14421.405,E2 14421.405} C_VEL
LIN {X 0,Y 309.667,Z 310.782,A -85,B 0,C 180,E1 14420.55,E2 14420.55} C_VEL
LIN {X 0,Y 315.489,Z 226.103,A -85,B 0,C 180,E1 14418.016,E2 14418.016} C_VEL
LIN {X 0,Y 315.671,Z 220.222,A -85,B 0,C 180,E1 14417.81,E2 14417.81} C_VEL
LIN {X 0,Y 312.063,Z 193.866,A -85,B 0,C 180,E1 14416.067,E2 14416.067} C_VEL
LIN {X 0,Y 308.245,Z 171.07,A -85,B 0,C 180,E1 14414.272,E2 14414.272} C_VEL
LIN {X 0,Y 310.335,Z 162.307,A -85,B 0,C 180,E1 14412.517,E2 14412.517} C_VEL
LIN {X 0,Y 308.369,Z 151.627,A -85,B 0,C 180,E1 14409.142,E2 14409.142} C_VEL
LIN {X 0,Y 306.1,Z 142.067,A -85,B 0,C 180,E1 14405.624,E2 14405.624} C_VEL
LIN {X 0,Y 303.799,Z 133.982,A -85,B 0,C 180,E1 14402.075,E2 14402.075} C_VEL
LIN {X 0,Y 301.606,Z 126.917,A -85,B 0,C 180,E1 14398.291,E2 14398.291} C_VEL
LIN {X 0,Y 299.892,Z 122.526,A -85,B 0,C 180,E1 14395.219,E2 14395.219} C_VEL
LIN {X 0,Y 298.839,Z 119.519,A -85,B 0,C 180,E1 14392.696,E2 14392.696} C_VEL
LIN {X 0,Y 297.637,Z 116.092,A -85,B 0,C 180,E1 14388.765,E2 14388.765} C_VEL
LIN {X 0,Y 296.713,Z 114.449,A -85,B 0,C 180,E1 14383.557,E2 14383.557} C_VEL
LIN {X 0,Y 297.04,Z 114.893,A -85,B 0,C 180,E1 14379.509,E2 14379.509} C_VEL
LIN {X 0,Y 298.556,Z 117.206,A -85,B 0,C 180,E1 14374.829,E2 14374.829} C_VEL
LIN {X 0,Y 300.573,Z 121.89,A -85,B 0,C 180,E1 14370.507,E2 14370.507} C_VEL
LIN {X 0,Y 302.256,Z 125.902,A -85,B 0,C 180,E1 14367.82,E2 14367.82} C_VEL
LIN {X 0,Y 304.121,Z 130.517,A -85,B 0,C 180,E1 14365.279,E2 14365.279} C_VEL
LIN {X 0,Y 306.536,Z 136.74,A -85,B 0,C 180,E1 14362.414,E2 14362.414} C_VEL
LIN {X 0,Y 309.47,Z 145.063,A -85,B 0,C 180,E1 14359.26,E2 14359.26} C_VEL
LIN {X 0,Y 312.644,Z 155.366,A -85,B 0,C 180,E1 14356.02,E2 14356.02} C_VEL
LIN {X 0,Y 315.17,Z 164.648,A -85,B 0,C 180,E1 14353.605,E2 14353.605} C_VEL
LIN {X 0,Y 317.325,Z 186.796,A -85,B 0,C 180,E1 14352.421,E2 14352.421} C_VEL
LIN {X 0,Y 317.943,Z 198.597,A -85,B 0,C 180,E1 14351.915,E2 14351.915} C_VEL
LIN {X 0,Y 311.737,Z 327.59,A -85,B 0,C 180,E1 14348.877,E2 14348.877} C_VEL
LIN {X 0,Y 310.46,Z 349.753,A -85,B 0,C 180,E1 14348.278,E2 14348.278} C_VEL
LIN {X 0,Y 308.368,Z 367.786,A -85,B 0,C 180,E1 14347.501,E2 14347.501} C_VEL
LIN {X 0,Y 305.529,Z 384.908,A -85,B 0,C 180,E1 14346.44,E2 14346.44} C_VEL
LIN {X 0,Y 302.17,Z 401.596,A -85,B 0,C 180,E1 14345.038,E2 14345.038} C_VEL
LIN {X 0,Y 298.34,Z 418.16,A -85,B 0,C 180,E1 14343.228,E2 14343.228} C_VEL
LIN {X 0,Y 294.618,Z 432.925,A -85,B 0,C 180,E1 14341.18,E2 14341.18} C_VEL
LIN {X 0,Y 290.906,Z 446.909,A -85,B 0,C 180,E1 14338.764,E2 14338.764} C_VEL
LIN {X 0,Y 287.47,Z 459.824,A -85,B 0,C 180,E1 14335.993,E2 14335.993} C_VEL
LIN {X 0,Y 284.601,Z 471.235,A -85,B 0,C 180,E1 14332.954,E2 14332.954} C_VEL
LIN {X 0,Y 282.439,Z 481.226,A -85,B 0,C 180,E1 14329.653,E2 14329.653} C_VEL
LIN {X 0,Y 281.034,Z 490.186,A -85,B 0,C 180,E1 14325.901,E2 14325.901} C_VEL
LIN {X 0,Y 280.606,Z 497.062,A -85,B 0,C 180,E1 14322.137,E2 14322.137} C_VEL
LIN {X 0,Y 280.931,Z 502.059,A -85,B 0,C 180,E1 14318.34,E2 14318.34} C_VEL
LIN {X 0,Y 281.599,Z 504.933,A -85,B 0,C 180,E1 14314.89,E2 14314.89} C_VEL
LIN {X 0,Y 282.147,Z 506.148,A -85,B 0,C 180,E1 14311.626,E2 14311.626} C_VEL
LIN {X 0,Y 282.225,Z 505.95,A -85,B 0,C 180,E1 14308.784,E2 14308.784} C_VEL
LIN {X 0,Y 281.806,Z 504.295,A -85,B 0,C 180,E1 14305.558,E2 14305.558} C_VEL
LIN {X 0,Y 281.191,Z 501.007,A -85,B 0,C 180,E1 14302.236,E2 14302.236} C_VEL
LIN {X 0,Y 280.792,Z 495.754,A -85,B 0,C 180,E1 14298.708,E2 14298.708} C_VEL
LIN {X 0,Y 280.961,Z 488.57,A -85,B 0,C 180,E1 14295.156,E2 14295.156} C_VEL
LIN {X 0,Y 281.81,Z 479.852,A -85,B 0,C 180,E1 14291.809,E2 14291.809} C_VEL
LIN {X 0,Y 283.314,Z 469.684,A -85,B 0,C 180,E1 14288.687,E2 14288.687} C_VEL
LIN {X 0,Y 285.388,Z 458.106,A -85,B 0,C 180,E1 14285.803,E2 14285.803} C_VEL
LIN {X 0,Y 287.931,Z 445.066,A -85,B 0,C 180,E1 14283.167,E2 14283.167} C_VEL
LIN {X 0,Y 290.804,Z 430.366,A -85,B 0,C 180,E1 14280.778,E2 14280.778} C_VEL
LIN {X 0,Y 293.602,Z 415.426,A -85,B 0,C 180,E1 14278.829,E2 14278.829} C_VEL
LIN {X 0,Y 296.451,Z 398.731,A -85,B 0,C 180,E1 14277.113,E2 14277.113} C_VEL
LIN {X 0,Y 298.979,Z 381.447,A -85,B 0,C 180,E1 14275.762,E2 14275.762} C_VEL
LIN {X 0,Y 301.081,Z 363.467,A -85,B 0,C 180,E1 14274.747,E2 14274.747} C_VEL
LIN {X 0,Y 302.385,Z 345.057,A -85,B 0,C 180,E1 14274.064,E2 14274.064} C_VEL
LIN {X 0,Y 308.086,Z 179.572,A -85,B 0,C 180,E1 14270.237,E2 14270.237} C_VEL
LIN {X 0,Y 307.66,Z 158.712,A -85,B 0,C 180,E1 14269.585,E2 14269.585} C_VEL
LIN {X 0,Y 308.929,Z 148.576,A -85,B 0,C 180,E1 14268.753,E2 14268.753} C_VEL
LIN {X 0,Y 301.026,Z 128.064,A -85,B 0,C 180,E1 14265.707,E2 14265.707} C_VEL
LIN {X 0,Y 292.911,Z 109.158,A -85,B 0,C 180,E1 14262.5,E2 14262.5} C_VEL
LIN {X 0,Y 285.664,Z 94.019,A -85,B 0,C 180,E1 14259.57,E2 14259.57} C_VEL
LIN {X 0,Y 282.509,Z 87.177,A -85,B 0,C 180,E1 14258.14,E2 14258.14} C_VEL
LIN {X 0,Y 282.415,Z 86.632,A -85,B 0,C 180,E1 14257.769,E2 14257.769} C_VEL
LIN {X 0,Y 282.418,Z 86.614,A -85,B 0,C 180,E1 14252.963,E2 14252.963} C_VEL
LIN {X 0,Y 282.423,Z 86.605,A -85,B 0,C 180,E1 14248.32,E2 14248.32} C_VEL
LIN {X 0,Y 282.408,Z 86.603,A -85,B 0,C 180,E1 14243.517,E2 14243.517} C_VEL
LIN {X 0,Y 282.42,Z 86.602,A -85,B 0,C 180,E1 14238.794,E2 14238.794} C_VEL
LIN {X 0,Y 282.4,Z 86.604,A -85,B 0,C 180,E1 14234.053,E2 14234.053} C_VEL
LIN {X 0,Y 282.409,Z 86.601,A -85,B 0,C 180,E1 14229.373,E2 14229.373} C_VEL
LIN {X 0,Y 282.411,Z 86.601,A -85,B 0,C 180,E1 14224.874,E2 14224.874} C_VEL
LIN {X 0,Y 282.395,Z 86.603,A -85,B 0,C 180,E1 14220.202,E2 14220.202} C_VEL
LIN {X 0,Y 282.407,Z 86.605,A -85,B 0,C 180,E1 14215.532,E2 14215.532} C_VEL
LIN {X 0,Y 282.405,Z 86.605,A -85,B 0,C 180,E1 14211.026,E2 14211.026} C_VEL
LIN {X 0,Y 282.39,Z 86.606,A -85,B 0,C 180,E1 14206.277,E2 14206.277} C_VEL
LIN {X 0,Y 282.411,Z 86.605,A -85,B 0,C 180,E1 14201.585,E2 14201.585} C_VEL
LIN {X 0,Y 282.387,Z 86.573,A -85,B 0,C 180,E1 14197.007,E2 14197.007} C_VEL
LIN {X 0,Y 282.401,Z 86.61,A -85,B 0,C 180,E1 14192.137,E2 14192.137} C_VEL
LIN {X 0,Y 282.405,Z 86.604,A -85,B 0,C 180,E1 14187.681,E2 14187.681} C_VEL
LIN {X 0,Y 282.446,Z 86.923,A -85,B 0,C 180,E1 14186.113,E2 14186.113} C_VEL
LIN {X 0,Y 283.921,Z 90.408,A -85,B 0,C 180,E1 14185.134,E2 14185.134} C_VEL
LIN {X 0,Y 284.968,Z 92.193,A -85,B 0,C 180,E1 14184.624,E2 14184.624} C_VEL
LIN {X 0,Y 290.844,Z 104.306,A -85,B 0,C 180,E1 14181.519,E2 14181.519} C_VEL
LIN {X 0,Y 296.578,Z 118.062,A -85,B 0,C 180,E1 14178.382,E2 14178.382} C_VEL
LIN {X 0,Y 301.404,Z 131.861,A -85,B 0,C 180,E1 14175.576,E2 14175.576} C_VEL
LIN {X 0,Y 305.085,Z 145.167,A -85,B 0,C 180,E1 14173.111,E2 14173.111} C_VEL
LIN {X 0,Y 302.964,Z 180.535,A -85,B 0,C 180,E1 14168.588,E2 14168.588} C_VEL
LIN {X 0,Y 301.336,Z 212.369,A -85,B 0,C 180,E1 14164.677,E2 14164.677} C_VEL
LIN {X 0,Y 302.031,Z 218.497,A -85,B 0,C 180,E1 14164.425,E2 14164.425} C_VEL
LIN {X 0,Y 299.109,Z 312.396,A -85,B 0,C 180,E1 14162.193,E2 14162.193} C_VEL
LIN {X 0,Y 298.951,Z 330.267,A -85,B 0,C 180,E1 14161.616,E2 14161.616} C_VEL
LIN {X 0,Y 298.305,Z 344.186,A -85,B 0,C 180,E1 14160.85,E2 14160.85} C_VEL
LIN {X 0,Y 297.012,Z 358.875,A -85,B 0,C 180,E1 14159.658,E2 14159.658} C_VEL
LIN {X 0,Y 295.294,Z 372.061,A -85,B 0,C 180,E1 14158.184,E2 14158.184} C_VEL
LIN {X 0,Y 293.433,Z 383.519,A -85,B 0,C 180,E1 14156.509,E2 14156.509} C_VEL
LIN {X 0,Y 291.383,Z 394.124,A -85,B 0,C 180,E1 14154.53,E2 14154.53} C_VEL
LIN {X 0,Y 289.066,Z 404.387,A -85,B 0,C 180,E1 14152.027,E2 14152.027} C_VEL
LIN {X 0,Y 286.976,Z 412.673,A -85,B 0,C 180,E1 14149.327,E2 14149.327} C_VEL
LIN {X 0,Y 285.247,Z 418.993,A -85,B 0,C 180,E1 14146.493,E2 14146.493} C_VEL
LIN {X 0,Y 283.951,Z 423.379,A -85,B 0,C 180,E1 14143.621,E2 14143.621} C_VEL
LIN {X 0,Y 283.039,Z 426.121,A -85,B 0,C 180,E1 14140.583,E2 14140.583} C_VEL
LIN {X 0,Y 282.52,Z 427.048,A -85,B 0,C 180,E1 14137.318,E2 14137.318} C_VEL
LIN {X 0,Y 282.422,Z 425.939,A -85,B 0,C 180,E1 14134.059,E2 14134.059} C_VEL
LIN {X 0,Y 282.704,Z 423.023,A -85,B 0,C 180,E1 14131.012,E2 14131.012} C_VEL
LIN {X 0,Y 283.312,Z 418.573,A -85,B 0,C 180,E1 14128.178,E2 14128.178} C_VEL
LIN {X 0,Y 284.279,Z 412.235,A -85,B 0,C 180,E1 14125.359,E2 14125.359} C_VEL
LIN {X 0,Y 285.517,Z 404.31,A -85,B 0,C 180,E1 14122.756,E2 14122.756} C_VEL
LIN {X 0,Y 286.953,Z 394.798,A -85,B 0,C 180,E1 14120.371,E2 14120.371} C_VEL
LIN {X 0,Y 288.422,Z 384.189,A -85,B 0,C 180,E1 14118.298,E2 14118.298} C_VEL
LIN {X 0,Y 289.87,Z 371.907,A -85,B 0,C 180,E1 14116.433,E2 14116.433} C_VEL
LIN {X 0,Y 291.161,Z 358.249,A -85,B 0,C 180,E1 14114.87,E2 14114.87} C_VEL
LIN {X 0,Y 291.941,Z 348.837,A -85,B 0,C 180,E1 14113.995,E2 14113.995} C_VEL
LIN {X 0,Y 292.797,Z 348.019,A -85,B 0,C 180,E1 14113.635,E2 14113.635} C_VEL
LIN {X 0,Y 294.882,Z 349.213,A -85,B 0,C 180,E1 14113.248,E2 14113.248} C_VEL
LIN {X 0,Y 292.767,Z 364.501,A -85,B 0,C 180,E1 14111.48,E2 14111.48} C_VEL
LIN {X 0,Y 290.645,Z 378.006,A -85,B 0,C 180,E1 14109.457,E2 14109.457} C_VEL
LIN {X 0,Y 288.694,Z 389.376,A -85,B 0,C 180,E1 14107.322,E2 14107.322} C_VEL
LIN {X 0,Y 286.772,Z 399.884,A -85,B 0,C 180,E1 14104.825,E2 14104.825} C_VEL
LIN {X 0,Y 285.195,Z 408.598,A -85,B 0,C 180,E1 14102.206,E2 14102.206} C_VEL
LIN {X 0,Y 283.88,Z 416.071,A -85,B 0,C 180,E1 14099.25,E2 14099.25} C_VEL
LIN {X 0,Y 283.042,Z 421.543,A -85,B 0,C 180,E1 14096.315,E2 14096.315} C_VEL
LIN {X 0,Y 282.564,Z 425.582,A -85,B 0,C 180,E1 14093.018,E2 14093.018} C_VEL
LIN {X 0,Y 282.541,Z 427.615,A -85,B 0,C 180,E1 14089.853,E2 14089.853} C_VEL
LIN {X 0,Y 282.746,Z 427.98,A -85,B 0,C 180,E1 14087.797,E2 14087.797} C_VEL
LIN {X 0,Y 282.062,Z 427.994,A -85,B 0,C 180,E1 14086.227,E2 14086.227} C_VEL
LIN {X 0,Y 278.608,Z 427.348,A -85,B 0,C 180,E1 14083.457,E2 14083.457} C_VEL
LIN {X 0,Y 276.998,Z 425.958,A -85,B 0,C 180,E1 14081.43,E2 14081.43} C_VEL
LIN {X 0,Y 277.111,Z 425.129,A -85,B 0,C 180,E1 14080.644,E2 14080.644} C_VEL
LIN {X 0,Y 278.99,Z 420.476,A -85,B 0,C 180,E1 14077.536,E2 14077.536} C_VEL
LIN {X 0,Y 281.456,Z 413.972,A -85,B 0,C 180,E1 14074.494,E2 14074.494} C_VEL
LIN {X 0,Y 284.33,Z 405.769,A -85,B 0,C 180,E1 14071.678,E2 14071.678} C_VEL
LIN {X 0,Y 287.442,Z 396.212,A -85,B 0,C 180,E1 14069.143,E2 14069.143} C_VEL
LIN {X 0,Y 290.524,Z 385.69,A -85,B 0,C 180,E1 14066.953,E2 14066.953} C_VEL
LIN {X 0,Y 294.01,Z 372.314,A -85,B 0,C 180,E1 14064.768,E2 14064.768} C_VEL
LIN {X 0,Y 297,Z 358.874,A -85,B 0,C 180,E1 14063.059,E2 14063.059} C_VEL
LIN {X 0,Y 299.792,Z 343.759,A -85,B 0,C 180,E1 14061.569,E2 14061.569} C_VEL
LIN {X 0,Y 301.971,Z 328.244,A -85,B 0,C 180,E1 14060.438,E2 14060.438} C_VEL
LIN {X 0,Y 303.636,Z 311.412,A -85,B 0,C 180,E1 14059.575,E2 14059.575} C_VEL
LIN {X 0,Y 309.814,Z 225.321,A -85,B 0,C 180,E1 14056.967,E2 14056.967} C_VEL
LIN {X 0,Y 309.818,Z 221.344,A -85,B 0,C 180,E1 14056.801,E2 14056.801} C_VEL
LIN {X 0,Y 306.503,Z 195.647,A -85,B 0,C 180,E1 14055.031,E2 14055.031} C_VEL
LIN {X 0,Y 302.455,Z 170.828,A -85,B 0,C 180,E1 14052.991,E2 14052.991} C_VEL
LIN {X 0,Y 303.702,Z 165.901,A -85,B 0,C 180,E1 14051.971,E2 14051.971} C_VEL
LIN {X 0,Y 301.899,Z 155.494,A -85,B 0,C 180,E1 14048.571,E2 14048.571} C_VEL
LIN {X 0,Y 299.789,Z 146.138,A -85,B 0,C 180,E1 14044.975,E2 14044.975} C_VEL
LIN {X 0,Y 297.521,Z 137.873,A -85,B 0,C 180,E1 14041.156,E2 14041.156} C_VEL
LIN {X 0,Y 295.617,Z 131.834,A -85,B 0,C 180,E1 14037.674,E2 14037.674} C_VEL
LIN {X 0,Y 294.263,Z 128.068,A -85,B 0,C 180,E1 14034.932,E2 14034.932} C_VEL
LIN {X 0,Y 293.39,Z 125.34,A -85,B 0,C 180,E1 14032.56,E2 14032.56} C_VEL
LIN {X 0,Y 292.293,Z 122.009,A -85,B 0,C 180,E1 14028.557,E2 14028.557} C_VEL
LIN {X 0,Y 291.504,Z 120.512,A -85,B 0,C 180,E1 14023.46,E2 14023.46} C_VEL
LIN {X 0,Y 291.851,Z 120.978,A -85,B 0,C 180,E1 14019.547,E2 14019.547} C_VEL
LIN {X 0,Y 293.289,Z 123.169,A -85,B 0,C 180,E1 14014.993,E2 14014.993} C_VEL
LIN {X 0,Y 295.167,Z 127.587,A -85,B 0,C 180,E1 14010.805,E2 14010.805} C_VEL
LIN {X 0,Y 296.87,Z 131.954,A -85,B 0,C 180,E1 14007.85,E2 14007.85} C_VEL
LIN {X 0,Y 298.695,Z 136.495,A -85,B 0,C 180,E1 14005.315,E2 14005.315} C_VEL
LIN {X 0,Y 301.474,Z 143.954,A -85,B 0,C 180,E1 14001.912,E2 14001.912} C_VEL
LIN {X 0,Y 304.533,Z 153.405,A -85,B 0,C 180,E1 13998.455,E2 13998.455} C_VEL
LIN {X 0,Y 307.485,Z 164.025,A -85,B 0,C 180,E1 13995.251,E2 13995.251} C_VEL
LIN {X 0,Y 310.053,Z 169.496,A -85,B 0,C 180,E1 13994.425,E2 13994.425} C_VEL
LIN {X 0,Y 312.176,Z 196.196,A -85,B 0,C 180,E1 13993.04,E2 13993.04} C_VEL
LIN {X 0,Y 311.797,Z 206.807,A -85,B 0,C 180,E1 13992.741,E2 13992.741} C_VEL
LIN {X 0,Y 304.688,Z 344.893,A -85,B 0,C 180,E1 13989.39,E2 13989.39} C_VEL
LIN {X 0,Y 302.633,Z 363.607,A -85,B 0,C 180,E1 13988.634,E2 13988.634} C_VEL
LIN {X 0,Y 299.792,Z 380.998,A -85,B 0,C 180,E1 13987.615,E2 13987.615} C_VEL
LIN {X 0,Y 296.376,Z 397.824,A -85,B 0,C 180,E1 13986.265,E2 13986.265} C_VEL
LIN {X 0,Y 292.496,Z 414.199,A -85,B 0,C 180,E1 13984.531,E2 13984.531} C_VEL
LIN {X 0,Y 288.506,Z 429.244,A -85,B 0,C 180,E1 13982.493,E2 13982.493} C_VEL
LIN {X 0,Y 284.342,Z 444.098,A -85,B 0,C 180,E1 13979.957,E2 13979.957} C_VEL
LIN {X 0,Y 280.588,Z 457.315,A -85,B 0,C 180,E1 13977.138,E2 13977.138} C_VEL
LIN {X 0,Y 277.402,Z 469.004,A -85,B 0,C 180,E1 13974.036,E2 13974.036} C_VEL
LIN {X 0,Y 274.943,Z 479.177,A -85,B 0,C 180,E1 13970.657,E2 13970.657} C_VEL
LIN {X 0,Y 273.324,Z 487.881,A -85,B 0,C 180,E1 13967.018,E2 13967.018} C_VEL
LIN {X 0,Y 272.652,Z 495.024,A -85,B 0,C 180,E1 13963.143,E2 13963.143} C_VEL
LIN {X 0,Y 272.82,Z 500.217,A -85,B 0,C 180,E1 13959.281,E2 13959.281} C_VEL
LIN {X 0,Y 273.491,Z 503.415,A -85,B 0,C 180,E1 13955.666,E2 13955.666} C_VEL
LIN {X 0,Y 274.134,Z 504.897,A -85,B 0,C 180,E1 13952.301,E2 13952.301} C_VEL
LIN {X 0,Y 274.335,Z 504.957,A -85,B 0,C 180,E1 13949.375,E2 13949.375} C_VEL
LIN {X 0,Y 273.991,Z 503.656,A -85,B 0,C 180,E1 13946.235,E2 13946.235} C_VEL
LIN {X 0,Y 273.351,Z 500.7,A -85,B 0,C 180,E1 13942.858,E2 13942.858} C_VEL
LIN {X 0,Y 272.847,Z 495.677,A -85,B 0,C 180,E1 13939.14,E2 13939.14} C_VEL
LIN {X 0,Y 272.922,Z 489.006,A -85,B 0,C 180,E1 13935.576,E2 13935.576} C_VEL
LIN {X 0,Y 273.685,Z 480.656,A -85,B 0,C 180,E1 13932.131,E2 13932.131} C_VEL
LIN {X 0,Y 275.127,Z 470.886,A -85,B 0,C 180,E1 13928.915,E2 13928.915} C_VEL
LIN {X 0,Y 277.246,Z 459.299,A -85,B 0,C 180,E1 13925.841,E2 13925.841} C_VEL
LIN {X 0,Y 279.898,Z 446.142,A -85,B 0,C 180,E1 13923.023,E2 13923.023} C_VEL
LIN {X 0,Y 282.808,Z 431.933,A -85,B 0,C 180,E1 13920.568,E2 13920.568} C_VEL
LIN {X 0,Y 285.799,Z 416.702,A -85,B 0,C 180,E1 13918.467,E2 13918.467} C_VEL
LIN {X 0,Y 288.701,Z 400.476,A -85,B 0,C 180,E1 13916.709,E2 13916.709} C_VEL
LIN {X 0,Y 291.376,Z 383.233,A -85,B 0,C 180,E1 13915.278,E2 13915.278} C_VEL
LIN {X 0,Y 293.631,Z 365.152,A -85,B 0,C 180,E1 13914.189,E2 13914.189} C_VEL
LIN {X 0,Y 295.098,Z 346.968,A -85,B 0,C 180,E1 13913.448,E2 13913.448} C_VEL
LIN {X 0,Y 301.151,Z 179.602,A -85,B 0,C 180,E1 13909.471,E2 13909.471} C_VEL
LIN {X 0,Y 300.82,Z 158.496,A -85,B 0,C 180,E1 13908.784,E2 13908.784} C_VEL
LIN {X 0,Y 301.849,Z 151.284,A -85,B 0,C 180,E1 13908.185,E2 13908.185} C_VEL
LIN {X 0,Y 293.69,Z 130.044,A -85,B 0,C 180,E1 13904.92,E2 13904.92} C_VEL
LIN {X 0,Y 285.286,Z 110.586,A -85,B 0,C 180,E1 13901.483,E2 13901.483} C_VEL
LIN {X 0,Y 278.146,Z 95.605,A -85,B 0,C 180,E1 13898.454,E2 13898.454} C_VEL
LIN {X 0,Y 274.559,Z 88.113,A -85,B 0,C 180,E1 13896.762,E2 13896.762} C_VEL
LIN {X 0,Y 274.476,Z 87.602,A -85,B 0,C 180,E1 13896.166,E2 13896.166} C_VEL
LIN {X 0,Y 274.473,Z 87.596,A -85,B 0,C 180,E1 13891.394,E2 13891.394} C_VEL
LIN {X 0,Y 274.48,Z 87.6,A -85,B 0,C 180,E1 13886.619,E2 13886.619} C_VEL
LIN {X 0,Y 274.468,Z 87.607,A -85,B 0,C 180,E1 13881.737,E2 13881.737} C_VEL
LIN {X 0,Y 274.479,Z 87.607,A -85,B 0,C 180,E1 13876.943,E2 13876.943} C_VEL
LIN {X 0,Y 274.468,Z 87.607,A -85,B 0,C 180,E1 13872.411,E2 13872.411} C_VEL
LIN {X 0,Y 274.474,Z 87.606,A -85,B 0,C 180,E1 13867.535,E2 13867.535} C_VEL
LIN {X 0,Y 274.468,Z 87.605,A -85,B 0,C 180,E1 13862.714,E2 13862.714} C_VEL
LIN {X 0,Y 274.461,Z 87.608,A -85,B 0,C 180,E1 13857.912,E2 13857.912} C_VEL
LIN {X 0,Y 274.477,Z 87.606,A -85,B 0,C 180,E1 13853.095,E2 13853.095} C_VEL
LIN {X 0,Y 274.455,Z 87.61,A -85,B 0,C 180,E1 13848.228,E2 13848.228} C_VEL
LIN {X 0,Y 274.473,Z 87.605,A -85,B 0,C 180,E1 13843.492,E2 13843.492} C_VEL
LIN {X 0,Y 274.447,Z 87.586,A -85,B 0,C 180,E1 13838.634,E2 13838.634} C_VEL
LIN {X 0,Y 274.467,Z 87.588,A -85,B 0,C 180,E1 13833.845,E2 13833.845} C_VEL
LIN {X 0,Y 274.45,Z 87.571,A -85,B 0,C 180,E1 13829.287,E2 13829.287} C_VEL
LIN {X 0,Y 274.504,Z 87.852,A -85,B 0,C 180,E1 13827.94,E2 13827.94} C_VEL
LIN {X 0,Y 276.04,Z 91.497,A -85,B 0,C 180,E1 13826.842,E2 13826.842} C_VEL
LIN {X 0,Y 277.185,Z 93.343,A -85,B 0,C 180,E1 13826.254,E2 13826.254} C_VEL
LIN {X 0,Y 281.84,Z 102.734,A -85,B 0,C 180,E1 13823.668,E2 13823.668} C_VEL
LIN {X 0,Y 286.632,Z 113.052,A -85,B 0,C 180,E1 13821.064,E2 13821.064} C_VEL
LIN {X 0,Y 292.163,Z 127.186,A -85,B 0,C 180,E1 13817.873,E2 13817.873} C_VEL
LIN {X 0,Y 296.731,Z 141.737,A -85,B 0,C 180,E1 13814.958,E2 13814.958} C_VEL
LIN {X 0,Y 298.379,Z 149.085,A -85,B 0,C 180,E1 13813.629,E2 13813.629} C_VEL
LIN {X 0,Y 296.074,Z 184.706,A -85,B 0,C 180,E1 13809.038,E2 13809.038} C_VEL
LIN {X 0,Y 294.547,Z 213.578,A -85,B 0,C 180,E1 13805.473,E2 13805.473} C_VEL
LIN {X 0,Y 295.215,Z 219.673,A -85,B 0,C 180,E1 13805.216,E2 13805.216} C_VEL
LIN {X 0,Y 292.161,Z 312.848,A -85,B 0,C 180,E1 13802.956,E2 13802.956} C_VEL
LIN {X 0,Y 291.973,Z 331.227,A -85,B 0,C 180,E1 13802.354,E2 13802.354} C_VEL
LIN {X 0,Y 291.279,Z 345.297,A -85,B 0,C 180,E1 13801.564,E2 13801.564} C_VEL
LIN {X 0,Y 289.913,Z 359.985,A -85,B 0,C 180,E1 13800.346,E2 13800.346} C_VEL
LIN {X 0,Y 288.012,Z 373.816,A -85,B 0,C 180,E1 13798.756,E2 13798.756} C_VEL
LIN {X 0,Y 285.9,Z 385.95,A -85,B 0,C 180,E1 13796.899,E2 13796.899} C_VEL
LIN {X 0,Y 283.887,Z 395.682,A -85,B 0,C 180,E1 13794.999,E2 13794.999} C_VEL
LIN {X 0,Y 281.561,Z 405.446,A -85,B 0,C 180,E1 13792.55,E2 13792.55} C_VEL
LIN {X 0,Y 279.417,Z 413.5,A -85,B 0,C 180,E1 13789.872,E2 13789.872} C_VEL
LIN {X 0,Y 277.685,Z 419.514,A -85,B 0,C 180,E1 13787.171,E2 13787.171} C_VEL
LIN {X 0,Y 276.274,Z 424.091,A -85,B 0,C 180,E1 13784.245,E2 13784.245} C_VEL
LIN {X 0,Y 275.188,Z 427.164,A -85,B 0,C 180,E1 13780.889,E2 13780.889} C_VEL
LIN {X 0,Y 274.614,Z 428.143,A -85,B 0,C 180,E1 13777.53,E2 13777.53} C_VEL
LIN {X 0,Y 274.49,Z 427.089,A -85,B 0,C 180,E1 13774.176,E2 13774.176} C_VEL
LIN {X 0,Y 274.768,Z 424.236,A -85,B 0,C 180,E1 13771.041,E2 13771.041} C_VEL
LIN {X 0,Y 275.394,Z 419.855,A -85,B 0,C 180,E1 13768.126,E2 13768.126} C_VEL
LIN {X 0,Y 276.394,Z 413.586,A -85,B 0,C 180,E1 13765.226,E2 13765.226} C_VEL
LIN {X 0,Y 277.794,Z 405.049,A -85,B 0,C 180,E1 13762.346,E2 13762.346} C_VEL
LIN {X 0,Y 279.375,Z 395.027,A -85,B 0,C 180,E1 13759.805,E2 13759.805} C_VEL
LIN {X 0,Y 280.937,Z 384.094,A -85,B 0,C 180,E1 13757.669,E2 13757.669} C_VEL
LIN {X 0,Y 282.38,Z 372.197,A -85,B 0,C 180,E1 13755.857,E2 13755.857} C_VEL
LIN {X 0,Y 283.655,Z 359.295,A -85,B 0,C 180,E1 13754.355,E2 13754.355} C_VEL
LIN {X 0,Y 284.113,Z 355.339,A -85,B 0,C 180,E1 13753.909,E2 13753.909} C_VEL
LIN {X 0,Y 284.866,Z 354.75,A -85,B 0,C 180,E1 13753.586,E2 13753.586} C_VEL
LIN {X 0,Y 286.74,Z 355.633,A -85,B 0,C 180,E1 13753.228,E2 13753.228} C_VEL
LIN {X 0,Y 284.451,Z 370.643,A -85,B 0,C 180,E1 13751.269,E2 13751.269} C_VEL
LIN {X 0,Y 282.358,Z 382.987,A -85,B 0,C 180,E1 13749.206,E2 13749.206} C_VEL
LIN {X 0,Y 280.324,Z 394.072,A -85,B 0,C 180,E1 13746.898,E2 13746.898} C_VEL
LIN {X 0,Y 278.401,Z 404.122,A -85,B 0,C 180,E1 13744.241,E2 13744.241} C_VEL
LIN {X 0,Y 276.813,Z 412.608,A -85,B 0,C 180,E1 13741.37,E2 13741.37} C_VEL
LIN {X 0,Y 275.605,Z 419.457,A -85,B 0,C 180,E1 13738.26,E2 13738.26} C_VEL
LIN {X 0,Y 274.891,Z 424.344,A -85,B 0,C 180,E1 13735.175,E2 13735.175} C_VEL
LIN {X 0,Y 274.575,Z 427.597,A -85,B 0,C 180,E1 13731.866,E2 13731.866} C_VEL
LIN {X 0,Y 274.731,Z 429.071,A -85,B 0,C 180,E1 13728.518,E2 13728.518} C_VEL
LIN {X 0,Y 275.354,Z 428.664,A -85,B 0,C 180,E1 13725.214,E2 13725.214} C_VEL
LIN {X 0,Y 276.476,Z 426.568,A -85,B 0,C 180,E1 13721.994,E2 13721.994} C_VEL
LIN {X 0,Y 277.111,Z 425.129,A -85,B 0,C 180,E1 13720.644,E2 13720.644} C_VEL
LIN {X 0,Y 277.013,Z 423.333,A -85,B 0,C 180,E1 13719.078,E2 13719.078} C_VEL
LIN {X 0,Y 274.465,Z 419.306,A -85,B 0,C 180,E1 13715.975,E2 13715.975} C_VEL
LIN {X 0,Y 273.96,Z 416.067,A -85,B 0,C 180,E1 13714.246,E2 13714.246} C_VEL
LIN {X 0,Y 274.331,Z 414.576,A -85,B 0,C 180,E1 13713.629,E2 13713.629} C_VEL
LIN {X 0,Y 277.384,Z 406.347,A -85,B 0,C 180,E1 13710.788,E2 13710.788} C_VEL
LIN {X 0,Y 280.799,Z 396.408,A -85,B 0,C 180,E1 13708.14,E2 13708.14} C_VEL
LIN {X 0,Y 284.286,Z 385.067,A -85,B 0,C 180,E1 13705.791,E2 13705.791} C_VEL
LIN {X 0,Y 287.665,Z 372.774,A -85,B 0,C 180,E1 13703.778,E2 13703.778} C_VEL
LIN {X 0,Y 290.893,Z 358.834,A -85,B 0,C 180,E1 13702.003,E2 13702.003} C_VEL
LIN {X 0,Y 293.78,Z 343.757,A -85,B 0,C 180,E1 13700.522,E2 13700.522} C_VEL
LIN {X 0,Y 296.184,Z 327.056,A -85,B 0,C 180,E1 13699.32,E2 13699.32} C_VEL
LIN {X 0,Y 297.806,Z 310.667,A -85,B 0,C 180,E1 13698.505,E2 13698.505} C_VEL
LIN {X 0,Y 304.248,Z 223.486,A -85,B 0,C 180,E1 13695.805,E2 13695.805} C_VEL
LIN {X 0,Y 301.079,Z 197.566,A -85,B 0,C 180,E1 13693.969,E2 13693.969} C_VEL
LIN {X 0,Y 297.265,Z 173.356,A -85,B 0,C 180,E1 13691.902,E2 13691.902} C_VEL
LIN {X 0,Y 296.987,Z 170.19,A -85,B 0,C 180,E1 13691.561,E2 13691.561} C_VEL
LIN {X 0,Y 296.328,Z 164.309,A -85,B 0,C 180,E1 13689.713,E2 13689.713} C_VEL
LIN {X 0,Y 294.553,Z 154.856,A -85,B 0,C 180,E1 13686.236,E2 13686.236} C_VEL
LIN {X 0,Y 292.641,Z 146.862,A -85,B 0,C 180,E1 13682.742,E2 13682.742} C_VEL
LIN {X 0,Y 290.79,Z 140.195,A -85,B 0,C 180,E1 13679.212,E2 13679.212} C_VEL
LIN {X 0,Y 289.207,Z 134.759,A -85,B 0,C 180,E1 13675.638,E2 13675.638} C_VEL
LIN {X 0,Y 287.943,Z 131.16,A -85,B 0,C 180,E1 13672.418,E2 13672.418} C_VEL
LIN {X 0,Y 287.021,Z 128.03,A -85,B 0,C 180,E1 13668.547,E2 13668.547} C_VEL
LIN {X 0,Y 286.303,Z 126.581,A -85,B 0,C 180,E1 13663.36,E2 13663.36} C_VEL
LIN {X 0,Y 286.704,Z 127.124,A -85,B 0,C 180,E1 13659.377,E2 13659.377} C_VEL
LIN {X 0,Y 288.071,Z 129.356,A -85,B 0,C 180,E1 13654.946,E2 13654.946} C_VEL
LIN {X 0,Y 289.872,Z 133.765,A -85,B 0,C 180,E1 13650.773,E2 13650.773} C_VEL
LIN {X 0,Y 291.51,Z 138.005,A -85,B 0,C 180,E1 13647.884,E2 13647.884} C_VEL
LIN {X 0,Y 293.508,Z 142.964,A -85,B 0,C 180,E1 13645.089,E2 13645.089} C_VEL
LIN {X 0,Y 295.981,Z 150.252,A -85,B 0,C 180,E1 13641.816,E2 13641.816} C_VEL
LIN {X 0,Y 298.775,Z 159.225,A -85,B 0,C 180,E1 13638.501,E2 13638.501} C_VEL
LIN {X 0,Y 300.507,Z 165.15,A -85,B 0,C 180,E1 13636.7,E2 13636.7} C_VEL
LIN {X 0,Y 304.904,Z 173.423,A -85,B 0,C 180,E1 13635.359,E2 13635.359} C_VEL
LIN {X 0,Y 306.721,Z 199.271,A -85,B 0,C 180,E1 13634.004,E2 13634.004} C_VEL
LIN {X 0,Y 299.629,Z 329.755,A -85,B 0,C 180,E1 13630.812,E2 13630.812} C_VEL
LIN {X 0,Y 298.236,Z 349.841,A -85,B 0,C 180,E1 13630.226,E2 13630.226} C_VEL
LIN {X 0,Y 295.825,Z 367.948,A -85,B 0,C 180,E1 13629.39,E2 13629.39} C_VEL
LIN {X 0,Y 292.757,Z 384.524,A -85,B 0,C 180,E1 13628.309,E2 13628.309} C_VEL
LIN {X 0,Y 289.01,Z 401.257,A -85,B 0,C 180,E1 13626.834,E2 13626.834} C_VEL
LIN {X 0,Y 284.923,Z 417.186,A -85,B 0,C 180,E1 13625.014,E2 13625.014} C_VEL
LIN {X 0,Y 280.789,Z 431.795,A -85,B 0,C 180,E1 13622.892,E2 13622.892} C_VEL
LIN {X 0,Y 276.53,Z 446.026,A -85,B 0,C 180,E1 13620.292,E2 13620.292} C_VEL
LIN {X 0,Y 272.563,Z 459.034,A -85,B 0,C 180,E1 13617.295,E2 13617.295} C_VEL
LIN {X 0,Y 269.255,Z 470.489,A -85,B 0,C 180,E1 13614.006,E2 13614.006} C_VEL
LIN {X 0,Y 266.743,Z 480.491,A -85,B 0,C 180,E1 13610.403,E2 13610.403} C_VEL
LIN {X 0,Y 265.206,Z 488.689,A -85,B 0,C 180,E1 13606.652,E2 13606.652} C_VEL
LIN {X 0,Y 264.641,Z 495.357,A -85,B 0,C 180,E1 13602.66,E2 13602.66} C_VEL
LIN {X 0,Y 264.935,Z 500.071,A -85,B 0,C 180,E1 13598.684,E2 13598.684} C_VEL
LIN {X 0,Y 265.684,Z 502.843,A -85,B 0,C 180,E1 13594.967,E2 13594.967} C_VEL
LIN {X 0,Y 266.282,Z 503.916,A -85,B 0,C 180,E1 13591.723,E2 13591.723} C_VEL
LIN {X 0,Y 266.382,Z 503.619,A -85,B 0,C 180,E1 13588.711,E2 13588.711} C_VEL
LIN {X 0,Y 265.919,Z 501.968,A -85,B 0,C 180,E1 13585.473,E2 13585.473} C_VEL
LIN {X 0,Y 265.245,Z 498.654,A -85,B 0,C 180,E1 13581.984,E2 13581.984} C_VEL
LIN {X 0,Y 264.846,Z 493.33,A -85,B 0,C 180,E1 13578.239,E2 13578.239} C_VEL
LIN {X 0,Y 265.097,Z 486.043,A -85,B 0,C 180,E1 13574.469,E2 13574.469} C_VEL
LIN {X 0,Y 266.121,Z 477.203,A -85,B 0,C 180,E1 13570.923,E2 13570.923} C_VEL
LIN {X 0,Y 267.853,Z 466.881,A -85,B 0,C 180,E1 13567.622,E2 13567.622} C_VEL
LIN {X 0,Y 270.261,Z 454.766,A -85,B 0,C 180,E1 13564.515,E2 13564.515} C_VEL
LIN {X 0,Y 273.03,Z 441.698,A -85,B 0,C 180,E1 13561.812,E2 13561.812} C_VEL
LIN {X 0,Y 276.067,Z 427.341,A -85,B 0,C 180,E1 13559.414,E2 13559.414} C_VEL
LIN {X 0,Y 279.12,Z 412.088,A -85,B 0,C 180,E1 13557.379,E2 13557.379} C_VEL
LIN {X 0,Y 282.033,Z 396.003,A -85,B 0,C 180,E1 13555.692,E2 13555.692} C_VEL
LIN {X 0,Y 284.717,Z 378.617,A -85,B 0,C 180,E1 13554.304,E2 13554.304} C_VEL
LIN {X 0,Y 286.876,Z 360.609,A -85,B 0,C 180,E1 13553.288,E2 13553.288} C_VEL
LIN {X 0,Y 288.165,Z 342.464,A -85,B 0,C 180,E1 13552.611,E2 13552.611} C_VEL
LIN {X 0,Y 294.29,Z 180.677,A -85,B 0,C 180,E1 13548.705,E2 13548.705} C_VEL
LIN {X 0,Y 293.945,Z 158.995,A -85,B 0,C 180,E1 13548,E2 13548} C_VEL
LIN {X 0,Y 294.597,Z 153.48,A -85,B 0,C 180,E1 13547.517,E2 13547.517} C_VEL
LIN {X 0,Y 286.668,Z 132.805,A -85,B 0,C 180,E1 13544.232,E2 13544.232} C_VEL
LIN {X 0,Y 279.003,Z 114.956,A -85,B 0,C 180,E1 13540.981,E2 13540.981} C_VEL
LIN {X 0,Y 271.461,Z 99.193,A -85,B 0,C 180,E1 13537.692,E2 13537.692} C_VEL
LIN {X 0,Y 268.032,Z 92.341,A -85,B 0,C 180,E1 13536.114,E2 13536.114} C_VEL
LIN {X 0,Y 266.587,Z 88.955,A -85,B 0,C 180,E1 13535.281,E2 13535.281} C_VEL
LIN {X 0,Y 266.542,Z 88.59,A -85,B 0,C 180,E1 13534.241,E2 13534.241} C_VEL
LIN {X 0,Y 266.534,Z 88.595,A -85,B 0,C 180,E1 13529.434,E2 13529.434} C_VEL
LIN {X 0,Y 266.54,Z 88.586,A -85,B 0,C 180,E1 13524.606,E2 13524.606} C_VEL
LIN {X 0,Y 266.526,Z 88.583,A -85,B 0,C 180,E1 13519.732,E2 13519.732} C_VEL
LIN {X 0,Y 266.551,Z 88.578,A -85,B 0,C 180,E1 13514.778,E2 13514.778} C_VEL
LIN {X 0,Y 266.522,Z 88.58,A -85,B 0,C 180,E1 13509.937,E2 13509.937} C_VEL
LIN {X 0,Y 266.535,Z 88.579,A -85,B 0,C 180,E1 13505.165,E2 13505.165} C_VEL
LIN {X 0,Y 266.52,Z 88.58,A -85,B 0,C 180,E1 13500.429,E2 13500.429} C_VEL
LIN {X 0,Y 266.53,Z 88.581,A -85,B 0,C 180,E1 13495.481,E2 13495.481} C_VEL
LIN {X 0,Y 266.523,Z 88.582,A -85,B 0,C 180,E1 13490.934,E2 13490.934} C_VEL
LIN {X 0,Y 266.526,Z 88.581,A -85,B 0,C 180,E1 13485.886,E2 13485.886} C_VEL
LIN {X 0,Y 266.523,Z 88.586,A -85,B 0,C 180,E1 13481.178,E2 13481.178} C_VEL
LIN {X 0,Y 266.513,Z 88.545,A -85,B 0,C 180,E1 13476.256,E2 13476.256} C_VEL
LIN {X 0,Y 266.526,Z 88.571,A -85,B 0,C 180,E1 13471.547,E2 13471.547} C_VEL
LIN {X 0,Y 266.57,Z 88.837,A -85,B 0,C 180,E1 13469.951,E2 13469.951} C_VEL
LIN {X 0,Y 268.084,Z 92.431,A -85,B 0,C 180,E1 13468.773,E2 13468.773} C_VEL
LIN {X 0,Y 269.265,Z 94.045,A -85,B 0,C 180,E1 13468.177,E2 13468.177} C_VEL
LIN {X 0,Y 271.366,Z 98.01,A -85,B 0,C 180,E1 13466.953,E2 13466.953} C_VEL
LIN {X 0,Y 277.723,Z 111.038,A -85,B 0,C 180,E1 13463.299,E2 13463.299} C_VEL
LIN {X 0,Y 283.473,Z 124.68,A -85,B 0,C 180,E1 13459.939,E2 13459.939} C_VEL
LIN {X 0,Y 288.28,Z 138.596,A -85,B 0,C 180,E1 13456.9,E2 13456.9} C_VEL
LIN {X 0,Y 291.815,Z 151.893,A -85,B 0,C 180,E1 13454.342,E2 13454.342} C_VEL
LIN {X 0,Y 289.348,Z 187.229,A -85,B 0,C 180,E1 13449.735,E2 13449.735} C_VEL
LIN {X 0,Y 287.799,Z 214.669,A -85,B 0,C 180,E1 13446.313,E2 13446.313} C_VEL
LIN {X 0,Y 288.459,Z 220.854,A -85,B 0,C 180,E1 13446.044,E2 13446.044} C_VEL
LIN {X 0,Y 285.267,Z 313.275,A -85,B 0,C 180,E1 13443.758,E2 13443.758} C_VEL
LIN {X 0,Y 285.052,Z 332.042,A -85,B 0,C 180,E1 13443.134,E2 13443.134} C_VEL
LIN {X 0,Y 284.3,Z 346.411,A -85,B 0,C 180,E1 13442.312,E2 13442.312} C_VEL
LIN {X 0,Y 282.859,Z 361.1,A -85,B 0,C 180,E1 13441.068,E2 13441.068} C_VEL
LIN {X 0,Y 280.941,Z 374.41,A -85,B 0,C 180,E1 13439.511,E2 13439.511} C_VEL
LIN {X 0,Y 278.902,Z 385.738,A -85,B 0,C 180,E1 13437.776,E2 13437.776} C_VEL
LIN {X 0,Y 276.632,Z 396.339,A -85,B 0,C 180,E1 13435.702,E2 13435.702} C_VEL
LIN {X 0,Y 274.165,Z 406.187,A -85,B 0,C 180,E1 13433.193,E2 13433.193} C_VEL
LIN {X 0,Y 271.886,Z 414.33,A -85,B 0,C 180,E1 13430.446,E2 13430.446} C_VEL
LIN {X 0,Y 270.037,Z 420.425,A -85,B 0,C 180,E1 13427.673,E2 13427.673} C_VEL
LIN {X 0,Y 268.521,Z 425.063,A -85,B 0,C 180,E1 13424.665,E2 13424.665} C_VEL
LIN {X 0,Y 267.346,Z 428.198,A -85,B 0,C 180,E1 13421.212,E2 13421.212} C_VEL
LIN {X 0,Y 266.709,Z 429.232,A -85,B 0,C 180,E1 13417.754,E2 13417.754} C_VEL
LIN {X 0,Y 266.552,Z 428.353,A -85,B 0,C 180,E1 13414.516,E2 13414.516} C_VEL
LIN {X 0,Y 266.774,Z 425.945,A -85,B 0,C 180,E1 13411.502,E2 13411.502} C_VEL
LIN {X 0,Y 267.419,Z 421.512,A -85,B 0,C 180,E1 13408.284,E2 13408.284} C_VEL
LIN {X 0,Y 268.419,Z 415.42,A -85,B 0,C 180,E1 13405.298,E2 13405.298} C_VEL
LIN {X 0,Y 269.726,Z 407.813,A -85,B 0,C 180,E1 13402.544,E2 13402.544} C_VEL
LIN {X 0,Y 271.26,Z 398.719,A -85,B 0,C 180,E1 13400.022,E2 13400.022} C_VEL
LIN {X 0,Y 272.996,Z 387.474,A -85,B 0,C 180,E1 13397.627,E2 13397.627} C_VEL
LIN {X 0,Y 274.578,Z 375.462,A -85,B 0,C 180,E1 13395.662,E2 13395.662} C_VEL
LIN {X 0,Y 276.181,Z 361.387,A -85,B 0,C 180,E1 13393.866,E2 13393.866} C_VEL
LIN {X 0,Y 276.913,Z 360.843,A -85,B 0,C 180,E1 13393.533,E2 13393.533} C_VEL
LIN {X 0,Y 278.545,Z 361.756,A -85,B 0,C 180,E1 13393.176,E2 13393.176} C_VEL
LIN {X 0,Y 276.224,Z 375.8,A -85,B 0,C 180,E1 13391.133,E2 13391.133} C_VEL
LIN {X 0,Y 274.135,Z 387.311,A -85,B 0,C 180,E1 13389.023,E2 13389.023} C_VEL
LIN {X 0,Y 271.858,Z 398.994,A -85,B 0,C 180,E1 13386.32,E2 13386.32} C_VEL
LIN {X 0,Y 270.036,Z 408.119,A -85,B 0,C 180,E1 13383.619,E2 13383.619} C_VEL
LIN {X 0,Y 268.489,Z 416.152,A -85,B 0,C 180,E1 13380.555,E2 13380.555} C_VEL
LIN {X 0,Y 267.421,Z 422.218,A -85,B 0,C 180,E1 13377.424,E2 13377.424} C_VEL
LIN {X 0,Y 266.796,Z 426.776,A -85,B 0,C 180,E1 13374.047,E2 13374.047} C_VEL
LIN {X 0,Y 266.648,Z 429.396,A -85,B 0,C 180,E1 13370.675,E2 13370.675} C_VEL
LIN {X 0,Y 266.996,Z 430.285,A -85,B 0,C 180,E1 13367.223,E2 13367.223} C_VEL
LIN {X 0,Y 267.829,Z 429.373,A -85,B 0,C 180,E1 13363.902,E2 13363.902} C_VEL
LIN {X 0,Y 269.321,Z 426.507,A -85,B 0,C 180,E1 13360.395,E2 13360.395} C_VEL
LIN {X 0,Y 271.321,Z 421.992,A -85,B 0,C 180,E1 13357.184,E2 13357.184} C_VEL
LIN {X 0,Y 274.034,Z 415.323,A -85,B 0,C 180,E1 13353.935,E2 13353.935} C_VEL
LIN {X 0,Y 274.331,Z 414.576,A -85,B 0,C 180,E1 13353.629,E2 13353.629} C_VEL
LIN {X 0,Y 274.812,Z 411.074,A -85,B 0,C 180,E1 13352.186,E2 13352.186} C_VEL
LIN {X 0,Y 273.382,Z 402.901,A -85,B 0,C 180,E1 13348.869,E2 13348.869} C_VEL
LIN {X 0,Y 273.729,Z 398.498,A -85,B 0,C 180,E1 13347.534,E2 13347.534} C_VEL
LIN {X 0,Y 274.124,Z 397.083,A -85,B 0,C 180,E1 13347.188,E2 13347.188} C_VEL
LIN {X 0,Y 278.073,Z 384.895,A -85,B 0,C 180,E1 13344.652,E2 13344.652} C_VEL
LIN {X 0,Y 281.631,Z 372.326,A -85,B 0,C 180,E1 13342.62,E2 13342.62} C_VEL
LIN {X 0,Y 285.252,Z 357.361,A -85,B 0,C 180,E1 13340.734,E2 13340.734} C_VEL
LIN {X 0,Y 288.162,Z 342.322,A -85,B 0,C 180,E1 13339.302,E2 13339.302} C_VEL
LIN {X 0,Y 290.592,Z 325.9,A -85,B 0,C 180,E1 13338.144,E2 13338.144} C_VEL
LIN {X 0,Y 292.281,Z 308.44,A -85,B 0,C 180,E1 13337.321,E2 13337.321} C_VEL
LIN {X 0,Y 298.712,Z 224.969,A -85,B 0,C 180,E1 13334.725,E2 13334.725} C_VEL
LIN {X 0,Y 295.839,Z 199.507,A -85,B 0,C 180,E1 13332.852,E2 13332.852} C_VEL
LIN {X 0,Y 292.243,Z 175.756,A -85,B 0,C 180,E1 13330.759,E2 13330.759} C_VEL
LIN {X 0,Y 291.664,Z 173.673,A -85,B 0,C 180,E1 13330.494,E2 13330.494} C_VEL
LIN {X 0,Y 290.149,Z 169.906,A -85,B 0,C 180,E1 13329.722,E2 13329.722} C_VEL
LIN {X 0,Y 288.546,Z 160.352,A -85,B 0,C 180,E1 13326.167,E2 13326.167} C_VEL
LIN {X 0,Y 286.78,Z 152.318,A -85,B 0,C 180,E1 13322.598,E2 13322.598} C_VEL
LIN {X 0,Y 285.07,Z 145.682,A -85,B 0,C 180,E1 13318.996,E2 13318.996} C_VEL
LIN {X 0,Y 283.583,Z 140.323,A -85,B 0,C 180,E1 13315.349,E2 13315.349} C_VEL
LIN {X 0,Y 282.421,Z 136.819,A -85,B 0,C 180,E1 13312.064,E2 13312.064} C_VEL
LIN {X 0,Y 281.695,Z 133.962,A -85,B 0,C 180,E1 13308.328,E2 13308.328} C_VEL
LIN {X 0,Y 281.134,Z 132.647,A -85,B 0,C 180,E1 13303.045,E2 13303.045} C_VEL
LIN {X 0,Y 281.598,Z 133.35,A -85,B 0,C 180,E1 13298.985,E2 13298.985} C_VEL
LIN {X 0,Y 282.813,Z 135.324,A -85,B 0,C 180,E1 13295.121,E2 13295.121} C_VEL
LIN {X 0,Y 284.513,Z 139.607,A -85,B 0,C 180,E1 13290.99,E2 13290.99} C_VEL
LIN {X 0,Y 286.159,Z 144.046,A -85,B 0,C 180,E1 13287.921,E2 13287.921} C_VEL
LIN {X 0,Y 288.142,Z 149.247,A -85,B 0,C 180,E1 13284.978,E2 13284.978} C_VEL
LIN {X 0,Y 290.871,Z 157.596,A -85,B 0,C 180,E1 13281.273,E2 13281.273} C_VEL
LIN {X 0,Y 293.226,Z 165.388,A -85,B 0,C 180,E1 13278.52,E2 13278.52} C_VEL
LIN {X 0,Y 299.721,Z 176.928,A -85,B 0,C 180,E1 13276.386,E2 13276.386} C_VEL
LIN {X 0,Y 301.111,Z 196.718,A -85,B 0,C 180,E1 13275.273,E2 13275.273} C_VEL
LIN {X 0,Y 301.12,Z 202.829,A -85,B 0,C 180,E1 13275.034,E2 13275.034} C_VEL
LIN {X 0,Y 292.882,Z 343.658,A -85,B 0,C 180,E1 13271.484,E2 13271.484} C_VEL
LIN {X 0,Y 290.666,Z 362.128,A -85,B 0,C 180,E1 13270.719,E2 13270.719} C_VEL
LIN {X 0,Y 287.593,Z 379.419,A -85,B 0,C 180,E1 13269.682,E2 13269.682} C_VEL
LIN {X 0,Y 283.865,Z 396.114,A -85,B 0,C 180,E1 13268.312,E2 13268.312} C_VEL
LIN {X 0,Y 279.606,Z 412.367,A -85,B 0,C 180,E1 13266.542,E2 13266.542} C_VEL
LIN {X 0,Y 275.15,Z 427.48,A -85,B 0,C 180,E1 13264.423,E2 13264.423} C_VEL
LIN {X 0,Y 270.647,Z 441.796,A -85,B 0,C 180,E1 13261.891,E2 13261.891} C_VEL
LIN {X 0,Y 266.377,Z 454.998,A -85,B 0,C 180,E1 13258.962,E2 13258.962} C_VEL
LIN {X 0,Y 262.684,Z 466.672,A -85,B 0,C 180,E1 13255.718,E2 13255.718} C_VEL
LIN {X 0,Y 259.753,Z 476.841,A -85,B 0,C 180,E1 13252.164,E2 13252.164} C_VEL
LIN {X 0,Y 257.729,Z 485.532,A -85,B 0,C 180,E1 13248.316,E2 13248.316} C_VEL
LIN {X 0,Y 256.748,Z 492.76,A -85,B 0,C 180,E1 13244.145,E2 13244.145} C_VEL
LIN {X 0,Y 256.77,Z 497.885,A -85,B 0,C 180,E1 13240.094,E2 13240.094} C_VEL
LIN {X 0,Y 257.463,Z 501.143,A -85,B 0,C 180,E1 13236.188,E2 13236.188} C_VEL
LIN {X 0,Y 258.226,Z 502.626,A -85,B 0,C 180,E1 13232.591,E2 13232.591} C_VEL
LIN {X 0,Y 258.506,Z 502.673,A -85,B 0,C 180,E1 13229.558,E2 13229.558} C_VEL
LIN {X 0,Y 258.17,Z 501.479,A -85,B 0,C 180,E1 13226.449,E2 13226.449} C_VEL
LIN {X 0,Y 257.452,Z 498.6,A -85,B 0,C 180,E1 13222.863,E2 13222.863} C_VEL
LIN {X 0,Y 256.916,Z 493.729,A -85,B 0,C 180,E1 13219.008,E2 13219.008} C_VEL
LIN {X 0,Y 257.018,Z 486.915,A -85,B 0,C 180,E1 13215.124,E2 13215.124} C_VEL
LIN {X 0,Y 257.897,Z 478.548,A -85,B 0,C 180,E1 13211.465,E2 13211.465} C_VEL
LIN {X 0,Y 259.513,Z 468.74,A -85,B 0,C 180,E1 13208.057,E2 13208.057} C_VEL
LIN {X 0,Y 261.959,Z 456.665,A -85,B 0,C 180,E1 13204.694,E2 13204.694} C_VEL
LIN {X 0,Y 264.776,Z 443.901,A -85,B 0,C 180,E1 13201.836,E2 13201.836} C_VEL
LIN {X 0,Y 267.955,Z 429.599,A -85,B 0,C 180,E1 13199.258,E2 13199.258} C_VEL
LIN {X 0,Y 271.198,Z 414.146,A -85,B 0,C 180,E1 13197.06,E2 13197.06} C_VEL
LIN {X 0,Y 274.339,Z 397.67,A -85,B 0,C 180,E1 13195.226,E2 13195.226} C_VEL
LIN {X 0,Y 277.112,Z 380.702,A -85,B 0,C 180,E1 13193.786,E2 13193.786} C_VEL
LIN {X 0,Y 279.443,Z 362.908,A -85,B 0,C 180,E1 13192.693,E2 13192.693} C_VEL
LIN {X 0,Y 280.946,Z 344.601,A -85,B 0,C 180,E1 13191.936,E2 13191.936} C_VEL
LIN {X 0,Y 287.429,Z 180.691,A -85,B 0,C 180,E1 13187.879,E2 13187.879} C_VEL
LIN {X 0,Y 287.225,Z 158.521,A -85,B 0,C 180,E1 13187.116,E2 13187.116} C_VEL
LIN {X 0,Y 287.532,Z 156.195,A -85,B 0,C 180,E1 13186.907,E2 13186.907} C_VEL
LIN {X 0,Y 279.832,Z 135.974,A -85,B 0,C 180,E1 13183.598,E2 13183.598} C_VEL
LIN {X 0,Y 271.828,Z 117.297,A -85,B 0,C 180,E1 13180.068,E2 13180.068} C_VEL
LIN {X 0,Y 264.439,Z 101.799,A -85,B 0,C 180,E1 13176.684,E2 13176.684} C_VEL
LIN {X 0,Y 260.183,Z 93.445,A -85,B 0,C 180,E1 13174.663,E2 13174.663} C_VEL
LIN {X 0,Y 258.649,Z 89.952,A -85,B 0,C 180,E1 13173.73,E2 13173.73} C_VEL
LIN {X 0,Y 258.603,Z 89.575,A -85,B 0,C 180,E1 13172.508,E2 13172.508} C_VEL
LIN {X 0,Y 258.592,Z 89.571,A -85,B 0,C 180,E1 13167.644,E2 13167.644} C_VEL
LIN {X 0,Y 258.611,Z 89.569,A -85,B 0,C 180,E1 13162.744,E2 13162.744} C_VEL
LIN {X 0,Y 258.586,Z 89.576,A -85,B 0,C 180,E1 13157.786,E2 13157.786} C_VEL
LIN {X 0,Y 258.601,Z 89.575,A -85,B 0,C 180,E1 13152.958,E2 13152.958} C_VEL
LIN {X 0,Y 258.584,Z 89.577,A -85,B 0,C 180,E1 13148.001,E2 13148.001} C_VEL
LIN {X 0,Y 258.594,Z 89.576,A -85,B 0,C 180,E1 13143.103,E2 13143.103} C_VEL
LIN {X 0,Y 258.578,Z 89.579,A -85,B 0,C 180,E1 13138.227,E2 13138.227} C_VEL
LIN {X 0,Y 258.606,Z 89.58,A -85,B 0,C 180,E1 13133.339,E2 13133.339} C_VEL
LIN {X 0,Y 258.576,Z 89.588,A -85,B 0,C 180,E1 13128.4,E2 13128.4} C_VEL
LIN {X 0,Y 258.596,Z 89.582,A -85,B 0,C 180,E1 13123.505,E2 13123.505} C_VEL
LIN {X 0,Y 258.571,Z 89.561,A -85,B 0,C 180,E1 13118.685,E2 13118.685} C_VEL
LIN {X 0,Y 258.589,Z 89.563,A -85,B 0,C 180,E1 13113.767,E2 13113.767} C_VEL
LIN {X 0,Y 258.624,Z 89.861,A -85,B 0,C 180,E1 13112.177,E2 13112.177} C_VEL
LIN {X 0,Y 260.321,Z 93.638,A -85,B 0,C 180,E1 13110.804,E2 13110.804} C_VEL
LIN {X 0,Y 261.463,Z 95.118,A -85,B 0,C 180,E1 13110.189,E2 13110.189} C_VEL
LIN {X 0,Y 263.492,Z 98.97,A -85,B 0,C 180,E1 13108.93,E2 13108.93} C_VEL
LIN {X 0,Y 268.353,Z 108.187,A -85,B 0,C 180,E1 13106.021,E2 13106.021} C_VEL
LIN {X 0,Y 274.223,Z 121.138,A -85,B 0,C 180,E1 13102.489,E2 13102.489} C_VEL
LIN {X 0,Y 279.245,Z 134.244,A -85,B 0,C 180,E1 13099.332,E2 13099.332} C_VEL
LIN {X 0,Y 283.697,Z 148.469,A -85,B 0,C 180,E1 13096.307,E2 13096.307} C_VEL
LIN {X 0,Y 285.218,Z 155.364,A -85,B 0,C 180,E1 13094.989,E2 13094.989} C_VEL
LIN {X 0,Y 282.698,Z 189.546,A -85,B 0,C 180,E1 13090.498,E2 13090.498} C_VEL
LIN {X 0,Y 281.1,Z 215.662,A -85,B 0,C 180,E1 13087.198,E2 13087.198} C_VEL
LIN {X 0,Y 281.768,Z 221.91,A -85,B 0,C 180,E1 13086.915,E2 13086.915} C_VEL
LIN {X 0,Y 278.432,Z 313.699,A -85,B 0,C 180,E1 13084.599,E2 13084.599} C_VEL
LIN {X 0,Y 278.181,Z 333.008,A -85,B 0,C 180,E1 13083.947,E2 13083.947} C_VEL
LIN {X 0,Y 277.374,Z 347.526,A -85,B 0,C 180,E1 13083.098,E2 13083.098} C_VEL
LIN {X 0,Y 275.852,Z 362.215,A -85,B 0,C 180,E1 13081.826,E2 13081.826} C_VEL
LIN {X 0,Y 273.857,Z 375.398,A -85,B 0,C 180,E1 13080.252,E2 13080.252} C_VEL
LIN {X 0,Y 271.679,Z 386.909,A -85,B 0,C 180,E1 13078.449,E2 13078.449} C_VEL
LIN {X 0,Y 269.187,Z 397.902,A -85,B 0,C 180,E1 13076.23,E2 13076.23} C_VEL
LIN {X 0,Y 266.608,Z 407.664,A -85,B 0,C 180,E1 13073.656,E2 13073.656} C_VEL
LIN {X 0,Y 264.198,Z 415.785,A -85,B 0,C 180,E1 13070.807,E2 13070.807} C_VEL
LIN {X 0,Y 262.277,Z 421.723,A -85,B 0,C 180,E1 13067.984,E2 13067.984} C_VEL
LIN {X 0,Y 260.664,Z 426.347,A -85,B 0,C 180,E1 13064.842,E2 13064.842} C_VEL
LIN {X 0,Y 259.451,Z 429.362,A -85,B 0,C 180,E1 13061.333,E2 13061.333} C_VEL
LIN {X 0,Y 258.786,Z 430.335,A -85,B 0,C 180,E1 13057.77,E2 13057.77} C_VEL
LIN {X 0,Y 258.631,Z 429.274,A -85,B 0,C 180,E1 13054.211,E2 13054.211} C_VEL
LIN {X 0,Y 258.931,Z 426.413,A -85,B 0,C 180,E1 13050.883,E2 13050.883} C_VEL
LIN {X 0,Y 259.619,Z 422.023,A -85,B 0,C 180,E1 13047.791,E2 13047.791} C_VEL
LIN {X 0,Y 260.72,Z 415.747,A -85,B 0,C 180,E1 13044.717,E2 13044.717} C_VEL
LIN {X 0,Y 262.262,Z 407.199,A -85,B 0,C 180,E1 13041.669,E2 13041.669} C_VEL
LIN {X 0,Y 263.932,Z 397.564,A -85,B 0,C 180,E1 13039.08,E2 13039.08} C_VEL
LIN {X 0,Y 265.633,Z 386.795,A -85,B 0,C 180,E1 13036.835,E2 13036.835} C_VEL
LIN {X 0,Y 267.224,Z 375.07,A -85,B 0,C 180,E1 13034.926,E2 13034.926} C_VEL
LIN {X 0,Y 268.231,Z 366.914,A -85,B 0,C 180,E1 13033.82,E2 13033.82} C_VEL
LIN {X 0,Y 268.948,Z 366.416,A -85,B 0,C 180,E1 13033.475,E2 13033.475} C_VEL
LIN {X 0,Y 270.331,Z 367.418,A -85,B 0,C 180,E1 13033.12,E2 13033.12} C_VEL
LIN {X 0,Y 267.81,Z 381.529,A -85,B 0,C 180,E1 13030.818,E2 13030.818} C_VEL
LIN {X 0,Y 265.546,Z 393.042,A -85,B 0,C 180,E1 13028.441,E2 13028.441} C_VEL
LIN {X 0,Y 263.275,Z 404.1,A -85,B 0,C 180,E1 13025.545,E2 13025.545} C_VEL
LIN {X 0,Y 261.443,Z 412.955,A -85,B 0,C 180,E1 13022.532,E2 13022.532} C_VEL
LIN {X 0,Y 260.096,Z 419.945,A -85,B 0,C 180,E1 13019.442,E2 13019.442} C_VEL
LIN {X 0,Y 259.203,Z 425.2,A -85,B 0,C 180,E1 13016.256,E2 13016.256} C_VEL
LIN {X 0,Y 258.746,Z 429.168,A -85,B 0,C 180,E1 13012.648,E2 13012.648} C_VEL
LIN {X 0,Y 258.808,Z 431.08,A -85,B 0,C 180,E1 13009.22,E2 13009.22} C_VEL
LIN {X 0,Y 259.375,Z 431.303,A -85,B 0,C 180,E1 13005.753,E2 13005.753} C_VEL
LIN {X 0,Y 260.426,Z 429.952,A -85,B 0,C 180,E1 13002.509,E2 13002.509} C_VEL
LIN {X 0,Y 262.186,Z 426.602,A -85,B 0,C 180,E1 12998.995,E2 12998.995} C_VEL
LIN {X 0,Y 264.628,Z 421.387,A -85,B 0,C 180,E1 12995.583,E2 12995.583} C_VEL
LIN {X 0,Y 267.608,Z 414.328,A -85,B 0,C 180,E1 12992.391,E2 12992.391} C_VEL
LIN {X 0,Y 271.022,Z 405.707,A -85,B 0,C 180,E1 12989.464,E2 12989.464} C_VEL
LIN {X 0,Y 274.124,Z 397.083,A -85,B 0,C 180,E1 12987.188,E2 12987.188} C_VEL
LIN {X 0,Y 274.987,Z 392.16,A -85,B 0,C 180,E1 12985.944,E2 12985.944} C_VEL
LIN {X 0,Y 274.379,Z 381.031,A -85,B 0,C 180,E1 12983.026,E2 12983.026} C_VEL
LIN {X 0,Y 274.904,Z 375.416,A -85,B 0,C 180,E1 12981.918,E2 12981.918} C_VEL
LIN {X 0,Y 275.311,Z 373.671,A -85,B 0,C 180,E1 12981.648,E2 12981.648} C_VEL
LIN {X 0,Y 278.98,Z 359.346,A -85,B 0,C 180,E1 12979.797,E2 12979.797} C_VEL
LIN {X 0,Y 282.058,Z 344.583,A -85,B 0,C 180,E1 12978.336,E2 12978.336} C_VEL
LIN {X 0,Y 284.718,Z 327.804,A -85,B 0,C 180,E1 12977.11,E2 12977.11} C_VEL
LIN {X 0,Y 286.518,Z 310.917,A -85,B 0,C 180,E1 12976.271,E2 12976.271} C_VEL
LIN {X 0,Y 293.364,Z 226.44,A -85,B 0,C 180,E1 12973.59,E2 12973.59} C_VEL
LIN {X 0,Y 290.69,Z 201.166,A -85,B 0,C 180,E1 12971.671,E2 12971.671} C_VEL
LIN {X 0,Y 287.612,Z 179.135,A -85,B 0,C 180,E1 12969.657,E2 12969.657} C_VEL
LIN {X 0,Y 283.237,Z 170.001,A -85,B 0,C 180,E1 12967.71,E2 12967.71} C_VEL
LIN {X 0,Y 281.662,Z 161.195,A -85,B 0,C 180,E1 12964.072,E2 12964.072} C_VEL
LIN {X 0,Y 279.965,Z 153.561,A -85,B 0,C 180,E1 12960.191,E2 12960.191} C_VEL
LIN {X 0,Y 278.472,Z 147.87,A -85,B 0,C 180,E1 12956.501,E2 12956.501} C_VEL
LIN {X 0,Y 277.599,Z 144.84,A -85,B 0,C 180,E1 12954.005,E2 12954.005} C_VEL
LIN {X 0,Y 277.038,Z 142.691,A -85,B 0,C 180,E1 12951.909,E2 12951.909} C_VEL
LIN {X 0,Y 276.382,Z 139.917,A -85,B 0,C 180,E1 12948.1,E2 12948.1} C_VEL
LIN {X 0,Y 275.962,Z 138.739,A -85,B 0,C 180,E1 12942.934,E2 12942.934} C_VEL
LIN {X 0,Y 276.435,Z 139.482,A -85,B 0,C 180,E1 12938.938,E2 12938.938} C_VEL
LIN {X 0,Y 277.589,Z 141.411,A -85,B 0,C 180,E1 12935.189,E2 12935.189} C_VEL
LIN {X 0,Y 279.108,Z 145.296,A -85,B 0,C 180,E1 12931.313,E2 12931.313} C_VEL
LIN {X 0,Y 280.663,Z 149.715,A -85,B 0,C 180,E1 12928.181,E2 12928.181} C_VEL
LIN {X 0,Y 282.564,Z 154.93,A -85,B 0,C 180,E1 12925.18,E2 12925.18} C_VEL
LIN {X 0,Y 285.033,Z 162.783,A -85,B 0,C 180,E1 12921.619,E2 12921.619} C_VEL
LIN {X 0,Y 286.08,Z 165.945,A -85,B 0,C 180,E1 12920.499,E2 12920.499} C_VEL
LIN {X 0,Y 292.482,Z 176.683,A -85,B 0,C 180,E1 12918.181,E2 12918.181} C_VEL
LIN {X 0,Y 294.988,Z 181.734,A -85,B 0,C 180,E1 12917.321,E2 12917.321} C_VEL
LIN {X 0,Y 295.98,Z 202.277,A -85,B 0,C 180,E1 12916.223,E2 12916.223} C_VEL
LIN {X 0,Y 287.213,Z 343.126,A -85,B 0,C 180,E1 12912.61,E2 12912.61} C_VEL
LIN {X 0,Y 284.846,Z 361.773,A -85,B 0,C 180,E1 12911.822,E2 12911.822} C_VEL
LIN {X 0,Y 281.662,Z 378.796,A -85,B 0,C 180,E1 12910.782,E2 12910.782} C_VEL
LIN {X 0,Y 277.849,Z 395.037,A -85,B 0,C 180,E1 12909.432,E2 12909.432} C_VEL
LIN {X 0,Y 273.384,Z 411.327,A -85,B 0,C 180,E1 12907.647,E2 12907.647} C_VEL
LIN {X 0,Y 268.679,Z 426.53,A -85,B 0,C 180,E1 12905.49,E2 12905.49} C_VEL
LIN {X 0,Y 263.935,Z 440.731,A -85,B 0,C 180,E1 12902.932,E2 12902.932} C_VEL
LIN {X 0,Y 259.539,Z 453.446,A -85,B 0,C 180,E1 12900.055,E2 12900.055} C_VEL
LIN {X 0,Y 255.538,Z 465.201,A -85,B 0,C 180,E1 12896.743,E2 12896.743} C_VEL
LIN {X 0,Y 252.312,Z 475.44,A -85,B 0,C 180,E1 12893.1,E2 12893.1} C_VEL
LIN {X 0,Y 250.032,Z 484.154,A -85,B 0,C 180,E1 12889.144,E2 12889.144} C_VEL
LIN {X 0,Y 248.843,Z 491.348,A -85,B 0,C 180,E1 12884.903,E2 12884.903} C_VEL
LIN {X 0,Y 248.738,Z 496.605,A -85,B 0,C 180,E1 12880.657,E2 12880.657} C_VEL
LIN {X 0,Y 249.395,Z 499.873,A -85,B 0,C 180,E1 12876.678,E2 12876.678} C_VEL
LIN {X 0,Y 250.227,Z 501.437,A -85,B 0,C 180,E1 12872.979,E2 12872.979} C_VEL
LIN {X 0,Y 250.593,Z 501.551,A -85,B 0,C 180,E1 12869.773,E2 12869.773} C_VEL
LIN {X 0,Y 250.262,Z 500.381,A -85,B 0,C 180,E1 12866.566,E2 12866.566} C_VEL
LIN {X 0,Y 249.437,Z 497.492,A -85,B 0,C 180,E1 12862.632,E2 12862.632} C_VEL
LIN {X 0,Y 248.956,Z 493.079,A -85,B 0,C 180,E1 12859.121,E2 12859.121} C_VEL
LIN {X 0,Y 249.07,Z 485.851,A -85,B 0,C 180,E1 12854.877,E2 12854.877} C_VEL
LIN {X 0,Y 250.016,Z 477.48,A -85,B 0,C 180,E1 12851.101,E2 12851.101} C_VEL
LIN {X 0,Y 251.731,Z 467.64,A -85,B 0,C 180,E1 12847.588,E2 12847.588} C_VEL
LIN {X 0,Y 254.309,Z 455.515,A -85,B 0,C 180,E1 12844.127,E2 12844.127} C_VEL
LIN {X 0,Y 257.26,Z 442.683,A -85,B 0,C 180,E1 12841.191,E2 12841.191} C_VEL
LIN {X 0,Y 260.584,Z 428.255,A -85,B 0,C 180,E1 12838.547,E2 12838.547} C_VEL
LIN {X 0,Y 263.965,Z 412.689,A -85,B 0,C 180,E1 12836.297,E2 12836.297} C_VEL
LIN {X 0,Y 267.229,Z 396.062,A -85,B 0,C 180,E1 12834.424,E2 12834.424} C_VEL
LIN {X 0,Y 270.108,Z 378.862,A -85,B 0,C 180,E1 12832.957,E2 12832.957} C_VEL
LIN {X 0,Y 272.482,Z 360.92,A -85,B 0,C 180,E1 12831.857,E2 12831.857} C_VEL
LIN {X 0,Y 273.941,Z 342.524,A -85,B 0,C 180,E1 12831.116,E2 12831.116} C_VEL
LIN {X 0,Y 280.625,Z 181.416,A -85,B 0,C 180,E1 12827.042,E2 12827.042} C_VEL
LIN {X 0,Y 280.419,Z 158.704,A -85,B 0,C 180,E1 12826.236,E2 12826.236} C_VEL
LIN {X 0,Y 272.918,Z 138.949,A -85,B 0,C 180,E1 12822.889,E2 12822.889} C_VEL
LIN {X 0,Y 265.105,Z 120.642,A -85,B 0,C 180,E1 12819.317,E2 12819.317} C_VEL
LIN {X 0,Y 258.198,Z 106.195,A -85,B 0,C 180,E1 12816.058,E2 12816.058} C_VEL
LIN {X 0,Y 252.421,Z 94.671,A -85,B 0,C 180,E1 12813.136,E2 12813.136} C_VEL
LIN {X 0,Y 250.717,Z 90.94,A -85,B 0,C 180,E1 12812.1,E2 12812.1} C_VEL
LIN {X 0,Y 250.665,Z 90.563,A -85,B 0,C 180,E1 12810.968,E2 12810.968} C_VEL
LIN {X 0,Y 250.654,Z 90.574,A -85,B 0,C 180,E1 12806.026,E2 12806.026} C_VEL
LIN {X 0,Y 250.666,Z 90.574,A -85,B 0,C 180,E1 12801.038,E2 12801.038} C_VEL
LIN {X 0,Y 250.648,Z 90.57,A -85,B 0,C 180,E1 12795.976,E2 12795.976} C_VEL
LIN {X 0,Y 250.658,Z 90.566,A -85,B 0,C 180,E1 12791.038,E2 12791.038} C_VEL
LIN {X 0,Y 250.643,Z 90.567,A -85,B 0,C 180,E1 12786.183,E2 12786.183} C_VEL
LIN {X 0,Y 250.661,Z 90.562,A -85,B 0,C 180,E1 12781.142,E2 12781.142} C_VEL
LIN {X 0,Y 250.64,Z 90.564,A -85,B 0,C 180,E1 12776.111,E2 12776.111} C_VEL
LIN {X 0,Y 250.656,Z 90.56,A -85,B 0,C 180,E1 12771.281,E2 12771.281} C_VEL
LIN {X 0,Y 250.639,Z 90.559,A -85,B 0,C 180,E1 12766.151,E2 12766.151} C_VEL
LIN {X 0,Y 250.65,Z 90.561,A -85,B 0,C 180,E1 12761.389,E2 12761.389} C_VEL
LIN {X 0,Y 250.636,Z 90.521,A -85,B 0,C 180,E1 12756.239,E2 12756.239} C_VEL
LIN {X 0,Y 250.674,Z 90.849,A -85,B 0,C 180,E1 12754.735,E2 12754.735} C_VEL
LIN {X 0,Y 252.14,Z 94.317,A -85,B 0,C 180,E1 12753.377,E2 12753.377} C_VEL
LIN {X 0,Y 253.768,Z 96.283,A -85,B 0,C 180,E1 12752.432,E2 12752.432} C_VEL
LIN {X 0,Y 255.854,Z 100.213,A -85,B 0,C 180,E1 12751.014,E2 12751.014} C_VEL
LIN {X 0,Y 259.515,Z 107.094,A -85,B 0,C 180,E1 12748.659,E2 12748.659} C_VEL
LIN {X 0,Y 263.553,Z 115.129,A -85,B 0,C 180,E1 12746.104,E2 12746.104} C_VEL
LIN {X 0,Y 268.664,Z 126.52,A -85,B 0,C 180,E1 12742.922,E2 12742.922} C_VEL
LIN {X 0,Y 273.523,Z 139.687,A -85,B 0,C 180,E1 12739.682,E2 12739.682} C_VEL
LIN {X 0,Y 277.577,Z 153.001,A -85,B 0,C 180,E1 12736.811,E2 12736.811} C_VEL
LIN {X 0,Y 278.781,Z 158.362,A -85,B 0,C 180,E1 12735.756,E2 12735.756} C_VEL
LIN {X 0,Y 275.99,Z 193.37,A -85,B 0,C 180,E1 12731.101,E2 12731.101} C_VEL
LIN {X 0,Y 274.485,Z 216.778,A -85,B 0,C 180,E1 12728.121,E2 12728.121} C_VEL
LIN {X 0,Y 275.142,Z 223.082,A -85,B 0,C 180,E1 12727.825,E2 12727.825} C_VEL
LIN {X 0,Y 271.663,Z 314.141,A -85,B 0,C 180,E1 12725.482,E2 12725.482} C_VEL
LIN {X 0,Y 271.37,Z 334.049,A -85,B 0,C 180,E1 12724.798,E2 12724.798} C_VEL
LIN {X 0,Y 270.504,Z 348.659,A -85,B 0,C 180,E1 12723.925,E2 12723.925} C_VEL
LIN {X 0,Y 268.897,Z 363.342,A -85,B 0,C 180,E1 12722.624,E2 12722.624} C_VEL
LIN {X 0,Y 266.8,Z 376.519,A -85,B 0,C 180,E1 12721.015,E2 12721.015} C_VEL
LIN {X 0,Y 264.505,Z 388.049,A -85,B 0,C 180,E1 12719.165,E2 12719.165} C_VEL
LIN {X 0,Y 262.01,Z 398.562,A -85,B 0,C 180,E1 12717.006,E2 12717.006} C_VEL
LIN {X 0,Y 259.276,Z 408.406,A -85,B 0,C 180,E1 12714.368,E2 12714.368} C_VEL
LIN {X 0,Y 256.695,Z 416.679,A -85,B 0,C 180,E1 12711.417,E2 12711.417} C_VEL
LIN {X 0,Y 254.665,Z 422.635,A -85,B 0,C 180,E1 12708.541,E2 12708.541} C_VEL
LIN {X 0,Y 252.925,Z 427.341,A -85,B 0,C 180,E1 12705.293,E2 12705.293} C_VEL
LIN {X 0,Y 251.618,Z 430.398,A -85,B 0,C 180,E1 12701.691,E2 12701.691} C_VEL
LIN {X 0,Y 250.886,Z 431.424,A -85,B 0,C 180,E1 12698.016,E2 12698.016} C_VEL
LIN {X 0,Y 250.693,Z 430.537,A -85,B 0,C 180,E1 12694.573,E2 12694.573} C_VEL
LIN {X 0,Y 250.931,Z 428.121,A -85,B 0,C 180,E1 12691.368,E2 12691.368} C_VEL
LIN {X 0,Y 251.639,Z 423.68,A -85,B 0,C 180,E1 12687.949,E2 12687.949} C_VEL
LIN {X 0,Y 252.742,Z 417.578,A -85,B 0,C 180,E1 12684.778,E2 12684.778} C_VEL
LIN {X 0,Y 254.184,Z 409.961,A -85,B 0,C 180,E1 12681.857,E2 12681.857} C_VEL
LIN {X 0,Y 255.874,Z 400.853,A -85,B 0,C 180,E1 12679.188,E2 12679.188} C_VEL
LIN {X 0,Y 257.784,Z 389.592,A -85,B 0,C 180,E1 12676.655,E2 12676.655} C_VEL
LIN {X 0,Y 259.626,Z 376.856,A -85,B 0,C 180,E1 12674.474,E2 12674.474} C_VEL
LIN {X 0,Y 260.364,Z 372.025,A -85,B 0,C 180,E1 12673.718,E2 12673.718} C_VEL
LIN {X 0,Y 261.284,Z 371.781,A -85,B 0,C 180,E1 12673.32,E2 12673.32} C_VEL
LIN {X 0,Y 262.147,Z 372.482,A -85,B 0,C 180,E1 12673.091,E2 12673.091} C_VEL
LIN {X 0,Y 259.638,Z 385.568,A -85,B 0,C 180,E1 12670.749,E2 12670.749} C_VEL
LIN {X 0,Y 257.189,Z 397.377,A -85,B 0,C 180,E1 12668.085,E2 12668.085} C_VEL
LIN {X 0,Y 254.885,Z 408.026,A -85,B 0,C 180,E1 12664.982,E2 12664.982} C_VEL
LIN {X 0,Y 253.187,Z 416.056,A -85,B 0,C 180,E1 12661.968,E2 12661.968} C_VEL
LIN {X 0,Y 251.799,Z 423.193,A -85,B 0,C 180,E1 12658.387,E2 12658.387} C_VEL
LIN {X 0,Y 251.045,Z 427.937,A -85,B 0,C 180,E1 12655.002,E2 12655.002} C_VEL
LIN {X 0,Y 250.782,Z 431.214,A -85,B 0,C 180,E1 12651.246,E2 12651.246} C_VEL
LIN {X 0,Y 251.069,Z 432.523,A -85,B 0,C 180,E1 12647.697,E2 12647.697} C_VEL
LIN {X 0,Y 251.964,Z 432.061,A -85,B 0,C 180,E1 12643.984,E2 12643.984} C_VEL
LIN {X 0,Y 253.465,Z 429.839,A -85,B 0,C 180,E1 12640.416,E2 12640.416} C_VEL
LIN {X 0,Y 255.771,Z 425.495,A -85,B 0,C 180,E1 12636.735,E2 12636.735} C_VEL
LIN {X 0,Y 258.438,Z 419.987,A -85,B 0,C 180,E1 12633.591,E2 12633.591} C_VEL
LIN {X 0,Y 261.89,Z 412.125,A -85,B 0,C 180,E1 12630.362,E2 12630.362} C_VEL
LIN {X 0,Y 265.482,Z 403.279,A -85,B 0,C 180,E1 12627.597,E2 12627.597} C_VEL
LIN {X 0,Y 269.577,Z 391.978,A -85,B 0,C 180,E1 12624.885,E2 12624.885} C_VEL
LIN {X 0,Y 273.428,Z 380.172,A -85,B 0,C 180,E1 12622.662,E2 12622.662} C_VEL
LIN {X 0,Y 275.311,Z 373.671,A -85,B 0,C 180,E1 12621.648,E2 12621.648} C_VEL
LIN {X 0,Y 276.223,Z 367.6,A -85,B 0,C 180,E1 12620.658,E2 12620.658} C_VEL
LIN {X 0,Y 275.685,Z 354.034,A -85,B 0,C 180,E1 12618.24,E2 12618.24} C_VEL
LIN {X 0,Y 276.034,Z 347.48,A -85,B 0,C 180,E1 12617.388,E2 12617.388} C_VEL
LIN {X 0,Y 276.349,Z 345.49,A -85,B 0,C 180,E1 12617.2,E2 12617.2} C_VEL
LIN {X 0,Y 279.165,Z 328.758,A -85,B 0,C 180,E1 12615.956,E2 12615.956} C_VEL
LIN {X 0,Y 281.052,Z 312.132,A -85,B 0,C 180,E1 12615.112,E2 12615.112} C_VEL
LIN {X 0,Y 288.15,Z 227.934,A -85,B 0,C 180,E1 12612.411,E2 12612.411} C_VEL
LIN {X 0,Y 285.77,Z 203.023,A -85,B 0,C 180,E1 12610.445,E2 12610.445} C_VEL
LIN {X 0,Y 283.235,Z 183.672,A -85,B 0,C 180,E1 12608.619,E2 12608.619} C_VEL
LIN {X 0,Y 278.493,Z 174.305,A -85,B 0,C 180,E1 12606.494,E2 12606.494} C_VEL
LIN {X 0,Y 276.301,Z 169.737,A -85,B 0,C 180,E1 12605.295,E2 12605.295} C_VEL
LIN {X 0,Y 274.867,Z 162.1,A -85,B 0,C 180,E1 12601.668,E2 12601.668} C_VEL
LIN {X 0,Y 273.513,Z 156.094,A -85,B 0,C 180,E1 12598.115,E2 12598.115} C_VEL
LIN {X 0,Y 272.454,Z 151.551,A -85,B 0,C 180,E1 12594.736,E2 12594.736} C_VEL
LIN {X 0,Y 271.594,Z 148.4,A -85,B 0,C 180,E1 12591.532,E2 12591.532} C_VEL
LIN {X 0,Y 271.134,Z 145.955,A -85,B 0,C 180,E1 12588.082,E2 12588.082} C_VEL
LIN {X 0,Y 270.788,Z 144.832,A -85,B 0,C 180,E1 12582.819,E2 12582.819} C_VEL
LIN {X 0,Y 271.29,Z 145.647,A -85,B 0,C 180,E1 12578.822,E2 12578.822} C_VEL
LIN {X 0,Y 272.366,Z 147.498,A -85,B 0,C 180,E1 12575.261,E2 12575.261} C_VEL
LIN {X 0,Y 273.78,Z 151.297,A -85,B 0,C 180,E1 12571.418,E2 12571.418} C_VEL
LIN {X 0,Y 275.328,Z 155.798,A -85,B 0,C 180,E1 12568.189,E2 12568.189} C_VEL
LIN {X 0,Y 277.373,Z 161.814,A -85,B 0,C 180,E1 12564.777,E2 12564.777} C_VEL
LIN {X 0,Y 278.797,Z 166.115,A -85,B 0,C 180,E1 12562.887,E2 12562.887} C_VEL
LIN {X 0,Y 284.03,Z 174.59,A -85,B 0,C 180,E1 12560.681,E2 12560.681} C_VEL
LIN {X 0,Y 289.151,Z 183.576,A -85,B 0,C 180,E1 12558.764,E2 12558.764} C_VEL
LIN {X 0,Y 290.234,Z 186.058,A -85,B 0,C 180,E1 12558.356,E2 12558.356} C_VEL
LIN {X 0,Y 290.844,Z 203.728,A -85,B 0,C 180,E1 12557.403,E2 12557.403} C_VEL
LIN {X 0,Y 281.676,Z 342.423,A -85,B 0,C 180,E1 12553.787,E2 12553.787} C_VEL
LIN {X 0,Y 279.224,Z 361.012,A -85,B 0,C 180,E1 12552.996,E2 12552.996} C_VEL
LIN {X 0,Y 275.932,Z 377.958,A -85,B 0,C 180,E1 12551.956,E2 12551.956} C_VEL
LIN {X 0,Y 271.96,Z 394.197,A -85,B 0,C 180,E1 12550.599,E2 12550.599} C_VEL
LIN {X 0,Y 267.517,Z 409.654,A -85,B 0,C 180,E1 12548.897,E2 12548.897} C_VEL
LIN {X 0,Y 262.547,Z 424.907,A -85,B 0,C 180,E1 12546.721,E2 12546.721} C_VEL
LIN {X 0,Y 257.514,Z 439.197,A -85,B 0,C 180,E1 12544.13,E2 12544.13} C_VEL
LIN {X 0,Y 252.81,Z 451.989,A -85,B 0,C 180,E1 12541.206,E2 12541.206} C_VEL
LIN {X 0,Y 248.486,Z 463.753,A -85,B 0,C 180,E1 12537.826,E2 12537.826} C_VEL
LIN {X 0,Y 244.949,Z 474.053,A -85,B 0,C 180,E1 12534.093,E2 12534.093} C_VEL
LIN {X 0,Y 242.387,Z 482.816,A -85,B 0,C 180,E1 12530.023,E2 12530.023} C_VEL
LIN {X 0,Y 240.962,Z 490.03,A -85,B 0,C 180,E1 12525.649,E2 12525.649} C_VEL
LIN {X 0,Y 240.719,Z 495.331,A -85,B 0,C 180,E1 12521.259,E2 12521.259} C_VEL
LIN {X 0,Y 241.382,Z 498.798,A -85,B 0,C 180,E1 12516.901,E2 12516.901} C_VEL
LIN {X 0,Y 242.274,Z 500.312,A -85,B 0,C 180,E1 12513.077,E2 12513.077} C_VEL
LIN {X 0,Y 242.679,Z 500.372,A -85,B 0,C 180,E1 12509.766,E2 12509.766} C_VEL
LIN {X 0,Y 242.308,Z 499.166,A -85,B 0,C 180,E1 12506.453,E2 12506.453} C_VEL
LIN {X 0,Y 241.46,Z 496.665,A -85,B 0,C 180,E1 12502.627,E2 12502.627} C_VEL
LIN {X 0,Y 240.958,Z 492.424,A -85,B 0,C 180,E1 12498.998,E2 12498.998} C_VEL
LIN {X 0,Y 241.041,Z 486.11,A -85,B 0,C 180,E1 12495.345,E2 12495.345} C_VEL
LIN {X 0,Y 241.967,Z 477.538,A -85,B 0,C 180,E1 12491.199,E2 12491.199} C_VEL
LIN {X 0,Y 243.672,Z 467.946,A -85,B 0,C 180,E1 12487.569,E2 12487.569} C_VEL
LIN {X 0,Y 246.064,Z 456.965,A -85,B 0,C 180,E1 12484.231,E2 12484.231} C_VEL
LIN {X 0,Y 249.006,Z 444.606,A -85,B 0,C 180,E1 12481.196,E2 12481.196} C_VEL
LIN {X 0,Y 252.446,Z 430.302,A -85,B 0,C 180,E1 12478.38,E2 12478.38} C_VEL
LIN {X 0,Y 255.898,Z 415.306,A -85,B 0,C 180,E1 12476.034,E2 12476.034} C_VEL
LIN {X 0,Y 259.209,Z 399.56,A -85,B 0,C 180,E1 12474.1,E2 12474.1} C_VEL
LIN {X 0,Y 262.319,Z 382.312,A -85,B 0,C 180,E1 12472.492,E2 12472.492} C_VEL
LIN {X 0,Y 264.897,Z 364.572,A -85,B 0,C 180,E1 12471.292,E2 12471.292} C_VEL
LIN {X 0,Y 266.652,Z 346.254,A -85,B 0,C 180,E1 12470.445,E2 12470.445} C_VEL
LIN {X 0,Y 268.519,Z 303.304,A -85,B 0,C 180,E1 12469.299,E2 12469.299} C_VEL
LIN {X 0,Y 273.861,Z 181.173,A -85,B 0,C 180,E1 12466.133,E2 12466.133} C_VEL
LIN {X 0,Y 273.494,Z 161.179,A -85,B 0,C 180,E1 12465.433,E2 12465.433} C_VEL
LIN {X 0,Y 271.715,Z 156.756,A -85,B 0,C 180,E1 12464.803,E2 12464.803} C_VEL
LIN {X 0,Y 264.454,Z 138.038,A -85,B 0,C 180,E1 12461.425,E2 12461.425} C_VEL
LIN {X 0,Y 256.98,Z 120.814,A -85,B 0,C 180,E1 12457.834,E2 12457.834} C_VEL
LIN {X 0,Y 250.361,Z 107.164,A -85,B 0,C 180,E1 12454.548,E2 12454.548} C_VEL
LIN {X 0,Y 244.705,Z 95.912,A -85,B 0,C 180,E1 12451.534,E2 12451.534} C_VEL
LIN {X 0,Y 242.882,Z 92.386,A -85,B 0,C 180,E1 12450.489,E2 12450.489} C_VEL
LIN {X 0,Y 242.722,Z 91.58,A -85,B 0,C 180,E1 12449.897,E2 12449.897} C_VEL
LIN {X 0,Y 242.723,Z 91.554,A -85,B 0,C 180,E1 12444.845,E2 12444.845} C_VEL
LIN {X 0,Y 242.713,Z 91.55,A -85,B 0,C 180,E1 12439.993,E2 12439.993} C_VEL
LIN {X 0,Y 242.734,Z 91.543,A -85,B 0,C 180,E1 12434.796,E2 12434.796} C_VEL
LIN {X 0,Y 242.712,Z 91.543,A -85,B 0,C 180,E1 12429.484,E2 12429.484} C_VEL
LIN {X 0,Y 242.711,Z 91.543,A -85,B 0,C 180,E1 12424.726,E2 12424.726} C_VEL
LIN {X 0,Y 242.717,Z 91.543,A -85,B 0,C 180,E1 12419.527,E2 12419.527} C_VEL
LIN {X 0,Y 242.701,Z 91.548,A -85,B 0,C 180,E1 12414.562,E2 12414.562} C_VEL
LIN {X 0,Y 242.712,Z 91.549,A -85,B 0,C 180,E1 12409.556,E2 12409.556} C_VEL
LIN {X 0,Y 242.697,Z 91.56,A -85,B 0,C 180,E1 12404.467,E2 12404.467} C_VEL
LIN {X 0,Y 242.715,Z 91.553,A -85,B 0,C 180,E1 12399.503,E2 12399.503} C_VEL
LIN {X 0,Y 242.778,Z 91.925,A -85,B 0,C 180,E1 12397.607,E2 12397.607} C_VEL
LIN {X 0,Y 244.306,Z 95.408,A -85,B 0,C 180,E1 12396.097,E2 12396.097} C_VEL
LIN {X 0,Y 246.044,Z 97.471,A -85,B 0,C 180,E1 12394.981,E2 12394.981} C_VEL
LIN {X 0,Y 248.079,Z 101.35,A -85,B 0,C 180,E1 12393.424,E2 12393.424} C_VEL
LIN {X 0,Y 249.095,Z 102.84,A -85,B 0,C 180,E1 12392.768,E2 12392.768} C_VEL
LIN {X 0,Y 252.289,Z 108.849,A -85,B 0,C 180,E1 12390.565,E2 12390.565} C_VEL
LIN {X 0,Y 255.958,Z 115.676,A -85,B 0,C 180,E1 12388.172,E2 12388.172} C_VEL
LIN {X 0,Y 261.316,Z 127.558,A -85,B 0,C 180,E1 12384.582,E2 12384.582} C_VEL
LIN {X 0,Y 266.369,Z 140.522,A -85,B 0,C 180,E1 12381.18,E2 12381.18} C_VEL
LIN {X 0,Y 270.466,Z 153.747,A -85,B 0,C 180,E1 12378.142,E2 12378.142} C_VEL
LIN {X 0,Y 272.347,Z 162.017,A -85,B 0,C 180,E1 12376.471,E2 12376.471} C_VEL
LIN {X 0,Y 269.335,Z 197.218,A -85,B 0,C 180,E1 12371.739,E2 12371.739} C_VEL
LIN {X 0,Y 267.916,Z 217.728,A -85,B 0,C 180,E1 12369.099,E2 12369.099} C_VEL
LIN {X 0,Y 268.592,Z 224.162,A -85,B 0,C 180,E1 12368.782,E2 12368.782} C_VEL
LIN {X 0,Y 264.961,Z 314.655,A -85,B 0,C 180,E1 12366.409,E2 12366.409} C_VEL
LIN {X 0,Y 264.621,Z 335.063,A -85,B 0,C 180,E1 12365.693,E2 12365.693} C_VEL
LIN {X 0,Y 263.692,Z 349.794,A -85,B 0,C 180,E1 12364.794,E2 12364.794} C_VEL
LIN {X 0,Y 262.001,Z 364.441,A -85,B 0,C 180,E1 12363.468,E2 12363.468} C_VEL
LIN {X 0,Y 259.794,Z 377.645,A -85,B 0,C 180,E1 12361.818,E2 12361.818} C_VEL
LIN {X 0,Y 257.478,Z 388.749,A -85,B 0,C 180,E1 12360.005,E2 12360.005} C_VEL
LIN {X 0,Y 254.883,Z 399.204,A -85,B 0,C 180,E1 12357.825,E2 12357.825} C_VEL
LIN {X 0,Y 251.988,Z 409.149,A -85,B 0,C 180,E1 12355.121,E2 12355.121} C_VEL
LIN {X 0,Y 249.482,Z 416.826,A -85,B 0,C 180,E1 12352.377,E2 12352.377} C_VEL
LIN {X 0,Y 247.235,Z 423.155,A -85,B 0,C 180,E1 12349.365,E2 12349.365} C_VEL
LIN {X 0,Y 245.203,Z 428.327,A -85,B 0,C 180,E1 12345.774,E2 12345.774} C_VEL
LIN {X 0,Y 243.795,Z 431.425,A -85,B 0,C 180,E1 12342.071,E2 12342.071} C_VEL
LIN {X 0,Y 243.023,Z 432.496,A -85,B 0,C 180,E1 12338.516,E2 12338.516} C_VEL
LIN {X 0,Y 242.765,Z 431.801,A -85,B 0,C 180,E1 12334.96,E2 12334.96} C_VEL
LIN {X 0,Y 242.994,Z 429.331,A -85,B 0,C 180,E1 12331.413,E2 12331.413} C_VEL
LIN {X 0,Y 243.717,Z 424.937,A -85,B 0,C 180,E1 12327.882,E2 12327.882} C_VEL
LIN {X 0,Y 244.862,Z 418.905,A -85,B 0,C 180,E1 12324.609,E2 12324.609} C_VEL
LIN {X 0,Y 246.362,Z 411.37,A -85,B 0,C 180,E1 12321.597,E2 12321.597} C_VEL
LIN {X 0,Y 248.124,Z 402.357,A -85,B 0,C 180,E1 12318.846,E2 12318.846} C_VEL
LIN {X 0,Y 250.115,Z 391.198,A -85,B 0,C 180,E1 12316.238,E2 12316.238} C_VEL
LIN {X 0,Y 251.938,Z 379.266,A -85,B 0,C 180,E1 12314.106,E2 12314.106} C_VEL
LIN {X 0,Y 252.479,Z 376.76,A -85,B 0,C 180,E1 12313.609,E2 12313.609} C_VEL
LIN {X 0,Y 253.304,Z 376.671,A -85,B 0,C 180,E1 12313.251,E2 12313.251} C_VEL
LIN {X 0,Y 253.959,Z 377.252,A -85,B 0,C 180,E1 12313.06,E2 12313.06} C_VEL
LIN {X 0,Y 251.326,Z 390.071,A -85,B 0,C 180,E1 12310.54,E2 12310.54} C_VEL
LIN {X 0,Y 248.696,Z 402.002,A -85,B 0,C 180,E1 12307.545,E2 12307.545} C_VEL
LIN {X 0,Y 246.599,Z 411.284,A -85,B 0,C 180,E1 12304.545,E2 12304.545} C_VEL
LIN {X 0,Y 244.858,Z 419.336,A -85,B 0,C 180,E1 12301.193,E2 12301.193} C_VEL
LIN {X 0,Y 243.653,Z 425.506,A -85,B 0,C 180,E1 12297.71,E2 12297.71} C_VEL
LIN {X 0,Y 242.976,Z 430.155,A -85,B 0,C 180,E1 12293.951,E2 12293.951} C_VEL
LIN {X 0,Y 242.874,Z 432.757,A -85,B 0,C 180,E1 12290.34,E2 12290.34} C_VEL
LIN {X 0,Y 243.326,Z 433.729,A -85,B 0,C 180,E1 12286.663,E2 12286.663} C_VEL
LIN {X 0,Y 244.415,Z 432.977,A -85,B 0,C 180,E1 12282.923,E2 12282.923} C_VEL
LIN {X 0,Y 246.234,Z 430.312,A -85,B 0,C 180,E1 12279.141,E2 12279.141} C_VEL
LIN {X 0,Y 248.753,Z 425.89,A -85,B 0,C 180,E1 12275.535,E2 12275.535} C_VEL
LIN {X 0,Y 251.891,Z 419.654,A -85,B 0,C 180,E1 12272.135,E2 12272.135} C_VEL
LIN {X 0,Y 255.497,Z 411.95,A -85,B 0,C 180,E1 12269.03,E2 12269.03} C_VEL
LIN {X 0,Y 259.51,Z 402.45,A -85,B 0,C 180,E1 12266.138,E2 12266.138} C_VEL
LIN {X 0,Y 263.864,Z 391.026,A -85,B 0,C 180,E1 12263.446,E2 12263.446} C_VEL
LIN {X 0,Y 268.041,Z 378.411,A -85,B 0,C 180,E1 12261.16,E2 12261.16} C_VEL
LIN {X 0,Y 272.056,Z 364.356,A -85,B 0,C 180,E1 12259.172,E2 12259.172} C_VEL
LIN {X 0,Y 275.618,Z 349.07,A -85,B 0,C 180,E1 12257.524,E2 12257.524} C_VEL
LIN {X 0,Y 276.349,Z 345.49,A -85,B 0,C 180,E1 12257.2,E2 12257.2} C_VEL
LIN {X 0,Y 276.962,Z 338.549,A -85,B 0,C 180,E1 12256.481,E2 12256.481} C_VEL
LIN {X 0,Y 275.681,Z 323.157,A -85,B 0,C 180,E1 12254.612,E2 12254.612} C_VEL
LIN {X 0,Y 275.539,Z 315.951,A -85,B 0,C 180,E1 12254.028,E2 12254.028} C_VEL
LIN {X 0,Y 275.68,Z 313.806,A -85,B 0,C 180,E1 12253.924,E2 12253.924} C_VEL
LIN {X 0,Y 283.167,Z 229.58,A -85,B 0,C 180,E1 12251.186,E2 12251.186} C_VEL
LIN {X 0,Y 280.996,Z 204.908,A -85,B 0,C 180,E1 12249.176,E2 12249.176} C_VEL
LIN {X 0,Y 279.034,Z 188.209,A -85,B 0,C 180,E1 12247.542,E2 12247.542} C_VEL
LIN {X 0,Y 274.54,Z 179.293,A -85,B 0,C 180,E1 12245.382,E2 12245.382} C_VEL
LIN {X 0,Y 271.534,Z 173.748,A -85,B 0,C 180,E1 12243.801,E2 12243.801} C_VEL
LIN {X 0,Y 269.37,Z 169.271,A -85,B 0,C 180,E1 12242.341,E2 12242.341} C_VEL
LIN {X 0,Y 268.12,Z 162.549,A -85,B 0,C 180,E1 12238.505,E2 12238.505} C_VEL
LIN {X 0,Y 267,Z 157.385,A -85,B 0,C 180,E1 12234.629,E2 12234.629} C_VEL
LIN {X 0,Y 266.218,Z 154.272,A -85,B 0,C 180,E1 12231.36,E2 12231.36} C_VEL
LIN {X 0,Y 265.82,Z 151.909,A -85,B 0,C 180,E1 12227.841,E2 12227.841} C_VEL
LIN {X 0,Y 265.612,Z 150.924,A -85,B 0,C 180,E1 12222.7,E2 12222.7} C_VEL
LIN {X 0,Y 266.144,Z 151.826,A -85,B 0,C 180,E1 12218.629,E2 12218.629} C_VEL
LIN {X 0,Y 267.115,Z 153.468,A -85,B 0,C 180,E1 12215.45,E2 12215.45} C_VEL
LIN {X 0,Y 268.471,Z 157.325,A -85,B 0,C 180,E1 12211.515,E2 12211.515} C_VEL
LIN {X 0,Y 270.247,Z 162.441,A -85,B 0,C 180,E1 12207.808,E2 12207.808} C_VEL
LIN {X 0,Y 271.643,Z 166.431,A -85,B 0,C 180,E1 12205.662,E2 12205.662} C_VEL
LIN {X 0,Y 276.911,Z 174.649,A -85,B 0,C 180,E1 12203.045,E2 12203.045} C_VEL
LIN {X 0,Y 282.134,Z 183.285,A -85,B 0,C 180,E1 12200.824,E2 12200.824} C_VEL
LIN {X 0,Y 285.589,Z 190.056,A -85,B 0,C 180,E1 12199.455,E2 12199.455} C_VEL
LIN {X 0,Y 285.951,Z 204.996,A -85,B 0,C 180,E1 12198.645,E2 12198.645} C_VEL
LIN {X 0,Y 276.355,Z 341.753,A -85,B 0,C 180,E1 12195.028,E2 12195.028} C_VEL
LIN {X 0,Y 273.769,Z 360.372,A -85,B 0,C 180,E1 12194.225,E2 12194.225} C_VEL
LIN {X 0,Y 270.329,Z 377.244,A -85,B 0,C 180,E1 12193.178,E2 12193.178} C_VEL
LIN {X 0,Y 266.19,Z 393.359,A -85,B 0,C 180,E1 12191.816,E2 12191.816} C_VEL
LIN {X 0,Y 261.298,Z 409.538,A -85,B 0,C 180,E1 12190.006,E2 12190.006} C_VEL
LIN {X 0,Y 256.105,Z 424.648,A -85,B 0,C 180,E1 12187.804,E2 12187.804} C_VEL
LIN {X 0,Y 250.623,Z 439.279,A -85,B 0,C 180,E1 12185.065,E2 12185.065} C_VEL
LIN {X 0,Y 245.52,Z 452.285,A -85,B 0,C 180,E1 12181.967,E2 12181.967} C_VEL
LIN {X 0,Y 240.99,Z 463.792,A -85,B 0,C 180,E1 12178.5,E2 12178.5} C_VEL
LIN {X 0,Y 237.263,Z 473.805,A -85,B 0,C 180,E1 12174.659,E2 12174.659} C_VEL
LIN {X 0,Y 234.435,Z 482.778,A -85,B 0,C 180,E1 12170.234,E2 12170.234} C_VEL
LIN {X 0,Y 232.967,Z 489.771,A -85,B 0,C 180,E1 12165.689,E2 12165.689} C_VEL
LIN {X 0,Y 232.746,Z 494.81,A -85,B 0,C 180,E1 12161.148,E2 12161.148} C_VEL
LIN {X 0,Y 233.496,Z 498.034,A -85,B 0,C 180,E1 12156.563,E2 12156.563} C_VEL
LIN {X 0,Y 234.411,Z 499.297,A -85,B 0,C 180,E1 12152.691,E2 12152.691} C_VEL
LIN {X 0,Y 234.762,Z 499.133,A -85,B 0,C 180,E1 12149.514,E2 12149.514} C_VEL
LIN {X 0,Y 234.23,Z 497.767,A -85,B 0,C 180,E1 12145.84,E2 12145.84} C_VEL
LIN {X 0,Y 233.432,Z 495.619,A -85,B 0,C 180,E1 12142.372,E2 12142.372} C_VEL
LIN {X 0,Y 232.949,Z 491.407,A -85,B 0,C 180,E1 12138.615,E2 12138.615} C_VEL
LIN {X 0,Y 233.067,Z 485.563,A -85,B 0,C 180,E1 12135.086,E2 12135.086} C_VEL
LIN {X 0,Y 234.603,Z 473.396,A -85,B 0,C 180,E1 12129.547,E2 12129.547} C_VEL
LIN {X 0,Y 236.715,Z 463.11,A -85,B 0,C 180,E1 12125.815,E2 12125.815} C_VEL
LIN {X 0,Y 239.54,Z 451.309,A -85,B 0,C 180,E1 12122.401,E2 12122.401} C_VEL
LIN {X 0,Y 242.808,Z 438.259,A -85,B 0,C 180,E1 12119.388,E2 12119.388} C_VEL
LIN {X 0,Y 246.364,Z 423.822,A -85,B 0,C 180,E1 12116.724,E2 12116.724} C_VEL
LIN {X 0,Y 249.842,Z 408.831,A -85,B 0,C 180,E1 12114.532,E2 12114.532} C_VEL
LIN {X 0,Y 253.179,Z 392.683,A -85,B 0,C 180,E1 12112.687,E2 12112.687} C_VEL
LIN {X 0,Y 256.187,Z 375.597,A -85,B 0,C 180,E1 12111.217,E2 12111.217} C_VEL
LIN {X 0,Y 258.592,Z 357.498,A -85,B 0,C 180,E1 12110.118,E2 12110.118} C_VEL
LIN {X 0,Y 260.025,Z 339.117,A -85,B 0,C 180,E1 12109.385,E2 12109.385} C_VEL
LIN {X 0,Y 267.14,Z 182.376,A -85,B 0,C 180,E1 12105.246,E2 12105.246} C_VEL
LIN {X 0,Y 266.772,Z 163.754,A -85,B 0,C 180,E1 12104.565,E2 12104.565} C_VEL
LIN {X 0,Y 264.398,Z 158.603,A -85,B 0,C 180,E1 12103.942,E2 12103.942} C_VEL
LIN {X 0,Y 257.251,Z 140.183,A -85,B 0,C 180,E1 12100.472,E2 12100.472} C_VEL
LIN {X 0,Y 250.014,Z 123.578,A -85,B 0,C 180,E1 12096.861,E2 12096.861} C_VEL
LIN {X 0,Y 243.425,Z 109.727,A -85,B 0,C 180,E1 12093.394,E2 12093.394} C_VEL
LIN {X 0,Y 238.774,Z 100.86,A -85,B 0,C 180,E1 12090.864,E2 12090.864} C_VEL
LIN {X 0,Y 236.644,Z 96.769,A -85,B 0,C 180,E1 12089.626,E2 12089.626} C_VEL
LIN {X 0,Y 234.879,Z 93.08,A -85,B 0,C 180,E1 12088.474,E2 12088.474} C_VEL
LIN {X 0,Y 234.782,Z 92.547,A -85,B 0,C 180,E1 12087.934,E2 12087.934} C_VEL
LIN {X 0,Y 234.793,Z 92.535,A -85,B 0,C 180,E1 12082.8,E2 12082.8} C_VEL
LIN {X 0,Y 234.773,Z 92.544,A -85,B 0,C 180,E1 12077.46,E2 12077.46} C_VEL
LIN {X 0,Y 234.777,Z 92.546,A -85,B 0,C 180,E1 12072.544,E2 12072.544} C_VEL
LIN {X 0,Y 234.796,Z 92.55,A -85,B 0,C 180,E1 12067.093,E2 12067.093} C_VEL
LIN {X 0,Y 234.771,Z 92.548,A -85,B 0,C 180,E1 12061.708,E2 12061.708} C_VEL
LIN {X 0,Y 234.769,Z 92.549,A -85,B 0,C 180,E1 12056.826,E2 12056.826} C_VEL
LIN {X 0,Y 234.775,Z 92.541,A -85,B 0,C 180,E1 12051.674,E2 12051.674} C_VEL
LIN {X 0,Y 234.757,Z 92.538,A -85,B 0,C 180,E1 12046.452,E2 12046.452} C_VEL
LIN {X 0,Y 234.79,Z 92.68,A -85,B 0,C 180,E1 12041.373,E2 12041.373} C_VEL
LIN {X 0,Y 235.03,Z 93.84,A -85,B 0,C 180,E1 12040.62,E2 12040.62} C_VEL
LIN {X 0,Y 236.84,Z 96.989,A -85,B 0,C 180,E1 12038.97,E2 12038.97} C_VEL
LIN {X 0,Y 238.255,Z 98.283,A -85,B 0,C 180,E1 12038.033,E2 12038.033} C_VEL
LIN {X 0,Y 240.027,Z 102.023,A -85,B 0,C 180,E1 12036.428,E2 12036.428} C_VEL
LIN {X 0,Y 241.362,Z 103.574,A -85,B 0,C 180,E1 12035.527,E2 12035.527} C_VEL
LIN {X 0,Y 243.696,Z 107.938,A -85,B 0,C 180,E1 12033.697,E2 12033.697} C_VEL
LIN {X 0,Y 247.135,Z 114.292,A -85,B 0,C 180,E1 12031.219,E2 12031.219} C_VEL
LIN {X 0,Y 251.314,Z 122.557,A -85,B 0,C 180,E1 12028.32,E2 12028.32} C_VEL
LIN {X 0,Y 256.05,Z 133.399,A -85,B 0,C 180,E1 12024.968,E2 12024.968} C_VEL
LIN {X 0,Y 260.779,Z 145.983,A -85,B 0,C 180,E1 12021.601,E2 12021.601} C_VEL
LIN {X 0,Y 264.746,Z 159.381,A -85,B 0,C 180,E1 12018.485,E2 12018.485} C_VEL
LIN {X 0,Y 266.014,Z 165.219,A -85,B 0,C 180,E1 12017.289,E2 12017.289} C_VEL
LIN {X 0,Y 262.721,Z 201.697,A -85,B 0,C 180,E1 12012.344,E2 12012.344} C_VEL
LIN {X 0,Y 261.45,Z 218.83,A -85,B 0,C 180,E1 12010.119,E2 12010.119} C_VEL
LIN {X 0,Y 262.119,Z 225.31,A -85,B 0,C 180,E1 12009.785,E2 12009.785} C_VEL
LIN {X 0,Y 258.334,Z 315.045,A -85,B 0,C 180,E1 12007.387,E2 12007.387} C_VEL
LIN {X 0,Y 257.948,Z 335.963,A -85,B 0,C 180,E1 12006.642,E2 12006.642} C_VEL
LIN {X 0,Y 257.017,Z 350.198,A -85,B 0,C 180,E1 12005.766,E2 12005.766} C_VEL
LIN {X 0,Y 255.249,Z 364.961,A -85,B 0,C 180,E1 12004.418,E2 12004.418} C_VEL
LIN {X 0,Y 252.992,Z 377.986,A -85,B 0,C 180,E1 12002.779,E2 12002.779} C_VEL
LIN {X 0,Y 250.512,Z 389.443,A -85,B 0,C 180,E1 12000.893,E2 12000.893} C_VEL
LIN {X 0,Y 247.543,Z 400.797,A -85,B 0,C 180,E1 11998.462,E2 11998.462} C_VEL
LIN {X 0,Y 244.511,Z 410.636,A -85,B 0,C 180,E1 11995.685,E2 11995.685} C_VEL
LIN {X 0,Y 241.683,Z 418.767,A -85,B 0,C 180,E1 11992.626,E2 11992.626} C_VEL
LIN {X 0,Y 239.361,Z 424.85,A -85,B 0,C 180,E1 11989.52,E2 11989.52} C_VEL
LIN {X 0,Y 237.428,Z 429.479,A -85,B 0,C 180,E1 11986.135,E2 11986.135} C_VEL
LIN {X 0,Y 235.91,Z 432.599,A -85,B 0,C 180,E1 11982.232,E2 11982.232} C_VEL
LIN {X 0,Y 235.068,Z 433.617,A -85,B 0,C 180,E1 11978.313,E2 11978.313} C_VEL
LIN {X 0,Y 234.836,Z 432.721,A -85,B 0,C 180,E1 11974.638,E2 11974.638} C_VEL
LIN {X 0,Y 235.088,Z 430.295,A -85,B 0,C 180,E1 11971.217,E2 11971.217} C_VEL
LIN {X 0,Y 235.867,Z 425.846,A -85,B 0,C 180,E1 11967.569,E2 11967.569} C_VEL
LIN {X 0,Y 237.088,Z 419.733,A -85,B 0,C 180,E1 11964.189,E2 11964.189} C_VEL
LIN {X 0,Y 238.682,Z 412.102,A -85,B 0,C 180,E1 11961.082,E2 11961.082} C_VEL
LIN {X 0,Y 240.548,Z 402.978,A -85,B 0,C 180,E1 11958.247,E2 11958.247} C_VEL
LIN {X 0,Y 242.557,Z 392.25,A -85,B 0,C 180,E1 11955.679,E2 11955.679} C_VEL
LIN {X 0,Y 244.421,Z 381.446,A -85,B 0,C 180,E1 11953.603,E2 11953.603} C_VEL
LIN {X 0,Y 245.322,Z 381.276,A -85,B 0,C 180,E1 11953.178,E2 11953.178} C_VEL
LIN {X 0,Y 245.719,Z 381.92,A -85,B 0,C 180,E1 11952.99,E2 11952.99} C_VEL
LIN {X 0,Y 242.961,Z 394.462,A -85,B 0,C 180,E1 11950.277,E2 11950.277} C_VEL
LIN {X 0,Y 240.398,Z 405.425,A -85,B 0,C 180,E1 11947.243,E2 11947.243} C_VEL
LIN {X 0,Y 238.347,Z 414.293,A -85,B 0,C 180,E1 11944.132,E2 11944.132} C_VEL
LIN {X 0,Y 236.654,Z 421.858,A -85,B 0,C 180,E1 11940.652,E2 11940.652} C_VEL
LIN {X 0,Y 235.551,Z 427.633,A -85,B 0,C 180,E1 11937.088,E2 11937.088} C_VEL
LIN {X 0,Y 234.991,Z 431.685,A -85,B 0,C 180,E1 11933.437,E2 11933.437} C_VEL
LIN {X 0,Y 235.01,Z 434.245,A -85,B 0,C 180,E1 11929.386,E2 11929.386} C_VEL
LIN {X 0,Y 235.651,Z 434.89,A -85,B 0,C 180,E1 11925.564,E2 11925.564} C_VEL
LIN {X 0,Y 237.091,Z 433.648,A -85,B 0,C 180,E1 11921.461,E2 11921.461} C_VEL
LIN {X 0,Y 239.132,Z 430.774,A -85,B 0,C 180,E1 11917.79,E2 11917.79} C_VEL
LIN {X 0,Y 242.163,Z 425.642,A -85,B 0,C 180,E1 11913.91,E2 11913.91} C_VEL
LIN {X 0,Y 245.555,Z 419.34,A -85,B 0,C 180,E1 11910.597,E2 11910.597} C_VEL
LIN {X 0,Y 249.745,Z 410.68,A -85,B 0,C 180,E1 11907.278,E2 11907.278} C_VEL
LIN {X 0,Y 254.074,Z 400.838,A -85,B 0,C 180,E1 11904.407,E2 11904.407} C_VEL
LIN {X 0,Y 258.616,Z 389.172,A -85,B 0,C 180,E1 11901.787,E2 11901.787} C_VEL
LIN {X 0,Y 263.009,Z 376.377,A -85,B 0,C 180,E1 11899.545,E2 11899.545} C_VEL
LIN {X 0,Y 267.196,Z 361.794,A -85,B 0,C 180,E1 11897.584,E2 11897.584} C_VEL
LIN {X 0,Y 270.607,Z 347.337,A -85,B 0,C 180,E1 11896.089,E2 11896.089} C_VEL
LIN {X 0,Y 273.57,Z 330.779,A -85,B 0,C 180,E1 11894.824,E2 11894.824} C_VEL
LIN {X 0,Y 275.647,Z 314.177,A -85,B 0,C 180,E1 11893.939,E2 11893.939} C_VEL
LIN {X 0,Y 275.68,Z 313.806,A -85,B 0,C 180,E1 11893.924,E2 11893.924} C_VEL
LIN {X 0,Y 275.718,Z 306.336,A -85,B 0,C 180,E1 11893.477,E2 11893.477} C_VEL
LIN {X 0,Y 273.601,Z 286.809,A -85,B 0,C 180,E1 11891.8,E2 11891.8} C_VEL
LIN {X 0,Y 273.763,Z 280.354,A -85,B 0,C 180,E1 11891.473,E2 11891.473} C_VEL
LIN {X 0,Y 278.317,Z 231.093,A -85,B 0,C 180,E1 11889.904,E2 11889.904} C_VEL
LIN {X 0,Y 276.439,Z 206.533,A -85,B 0,C 180,E1 11887.822,E2 11887.822} C_VEL
LIN {X 0,Y 274.967,Z 193.165,A -85,B 0,C 180,E1 11886.473,E2 11886.473} C_VEL
LIN {X 0,Y 271.211,Z 185.242,A -85,B 0,C 180,E1 11884.494,E2 11884.494} C_VEL
